      T     #OutTotalWeight;
      L     #Set001.RecipeNr;
      T     #OutRecipeNr;
      L     #Set001.Step;
      T     #OutLCStep;
//Reset old alarm flags with CmdFaultReset
      A     #Par.HelpFlags.OutFlagFaultResetDone;
      A     "SYS_Pulse1000ms";
      R     #Par.HelpFlags.OutFlagFaultResetDone;
      R     #Par.HelpFlags.OutFaultResetDone;
      S     #Par.HelpFlags.OutTestNewAlarm;
      L     0;
      L     #Set001.AlarmNr;
      ==I;
      =     #Par.HelpFlags.OutNoAlarm;
//  keep old alalrm number
      A     #Par.HelpFlags.OutNoAlarm;
      A     #Par.HelpFlags.OutRelevantFault;
      AN    #Par.HelpFlags.OutTestNewAlarm;
      AN    #InLocal;
      AN    #InManual;
      JC    rA1;
      T     #OutAlarmNr;
//--------------------------------------
//Calculate job weight on WtNotErasable
rA1:  L     #Set001.WtNotErasable;
//---  Init first, if old value < 0  ---
      L     #Par.OutNotErasableWeight;
      L     0;
      <D;
      JC    PgZ2;
//---  Calculate Weight ---
      L     #Set001.WtNotErasable;
      L     #Par.OutNotErasableWeight;
      -D;
      JM    PgZ1;
      JU    PgPo;
PgZ1: L     L#1000000000;	//[7.5] Overflow is 999999999
      +D;
      JM    PgZ2;	//[7.5]
PgPo: L     10000;	// Maximum change by relaod software
      >D;
      JC    PgZ2;
      TAK;
      L     #OutJobWeight;
      +D;
      T     #OutJobWeight;	//--> Total weight
PgZ2: L     #Set001.WtNotErasable;
      T     #Par.OutNotErasableWeight;
      JU    R11;	//[7.0]   
//===============================
//[7.0]--> LC Parameter 
//Reading dataset 11
R11:  L     "SYS_DirectCtrlLCDB".PC.ObjectNo;
      L     #Par.ParObjectNo;
      <>I;
      JC    R127;
      AN    "SYS_DirectCtrlLCDB".PC.Hsk.FExamineFirst;
      AN    "SYS_DirectCtrlLCDB".PC.Hsk.FExamineNext;
      JC    R127;
// -- Start Reading with Dataset 11
      L     11;
      T     #DPData.NrRcvDataSet;
      L     253;	//First
      A     "SYS_DirectCtrlLCDB".PC.Hsk.FExamineFirst;
      JC    rLC9;
      L     254;	//Next
rLC9: T     #DPData.IdxRcvDataSet;
      JU    rcv0;
//---Answer  dataset 11 ---
//---Answer  dataset 12 ---
r11:  L     #DPData.NrRcvDataSet;
      L     11;
      <>I;
      JC    rLCB;
// Answer Dataset 11
      L     '  ';
      T     "SYS_DirectCtrlLCDB".PC.Value[1];
      L     #DPData.Data[1];
      T     DB10.DBD 60;
      L     #DPData.Data[2];
      T     DB10.DBD 64;
      L     #DPData.Data[3];
      T     DB10.DBD 68;
      L     #DPData.Data[4];
      T     DB10.DBD 72;
      L     #DPData.IdxRcvDataSet;
      L     255;
      ==I;
      JC    rLCE;
      S     "SYS_DirectCtrlLCDB".GC.Set11Done;
      L     12;
      T     #DPData.NrRcvDataSet;
      L     0;
      T     #DPData.IdxRcvDataSet;
      JU    rcv0;	//--> Read dataset 12
// Answer Dataset 12
rLCB: L     #DPData.NrRcvDataSet;
      L     12;
      <>I;
      JC    r127;
      L     #DPData.Data[1];
      T     DB10.DBD 76;
      L     #DPData.Data[2];
      T     DB10.DBD 80;
      L     #DPData.Data[3];
      T     DB10.DBD 84;
      L     #DPData.Data[4];
      T     DB10.DBD 88;
      AN    "SYS_DirectCtrlLCDB".GC.Set11Done;
      JC    R127;
rLCE: L     12;
      CALL  "SYS_DirectCtrl";
      JU    R127;
//<--[7.0]
//===============================
//Answer  dataset 127
r127: L     #DPData.NrRcvDataSet;
      L     127;
      <>I;
      JC    r128;
      L     #DPData.Data[2];	//WtActual
      SRD   24;
      T     #tmpDecPoint;
      L     0;	//0 Decimal points == 1000gr
      ==I;
      L     1000;
      JC    rmul;
      L     #tmpDecPoint;
      L     1;	//1 Decimal points == 100gr
      ==I;
      L     100;
      JC    rmul;
      L     #tmpDecPoint;
      L     2;	//2 Decimal points == 10gr
      ==I;
      L     10;
      JC    rmul;
      L     1;	//3 Decimal points == 1gr
rmul: L     #DPData.Data[1];	//WtActual
      *D;
      T     #OutScaleWeight;
      JU    R128;
//===============================
//Answer  dataset 128
r128: L     #DPData.NrRcvDataSet;
      L     128;
      <>I;
      JC    r129;
      JU    R129;
//===============================
//Answer  dataset 129
r129: L     #DPData.NrRcvDataSet;
      L     129;
      <>I;
      JC    r136;
      S     #RecipeDiff.OutReadDone;
      R     #RecipeDiff.CmdRead;
      L     #DPData.Data[1];
      T     #DUMP.InDumpWeight;
      L     #DPData.Data[2];
      T     #DUMP.InFlowrateHighLimit;
      L     #DPData.Data[3];
      T     #DUMP.InFlowrateLowLimit;
      L     #DPData.Data[4];
      T     #DUMP.spare;
      JU    R001;
//===============================
//Answer  dataset 136
r136: L     #DPData.NrRcvDataSet;
      L     136;
      <>I;
      JC    R001;	// =no valide answer read dataset 001
      CALL  "SIEMENS_BLKMOV" (
           SRCBLK                   := #DPData.Data,
           RET_VAL                  := #tmpReturn,
           DSTBLK                   := #Set136);
      L     #RecipeDiff.InRecipeNr;
      L     #DPData.IdxRcvDataSet;
      ==I;
      JCN   R001;
      S     #RecipeDiff.OutReadDone;
      R     #RecipeDiff.CmdRead;
      L     #Set136.Density;
      T     #RecipeDiff.InOutDensity;
      L     #Set136.Factor;
      T     #RecipeDiff.InOutFactor;
      L     #Set136.AutoCorrFactor;
      T     #RecipeDiff.InOutAutoCorrFactor;
      L     #Set136.CutoffWt;
      T     #RecipeDiff.InOutCutoffWeight;
      JU    R001;
//===============================
//Read Dataset 001
R001: L     1;
      T     #DPData.NrRcvDataSet;
      L     0;
      T     #DPData.IdxRcvDataSet;
      A     #Par.HelpFlags.OutFaultResetDone;
      AN    "SYS_Pulse1000ms";
      S     #Par.HelpFlags.OutFlagFaultResetDone;
      JU    rcv0;
//===============================
//Read Dataset 127
R127: L     127;
      T     #DPData.NrRcvDataSet;
      L     0;
      T     #DPData.IdxRcvDataSet;
      JU    rcv0;
//===============================
//Read Dataset 128
R128: JU    R129;
      JU    rcv0;
//===============================
//Read Dataset 129
R129: AN    #RecipeDiff.CmdRead;
      ON    #Par.ParDUMP;
      JC    R136;
      L     129;
      T     #DPData.NrRcvDataSet;
      L     0;
      T     #DPData.IdxRcvDataSet;
      JU    rcv0;
//===============================
//Read Dataset 136
R136: AN    #RecipeDiff.CmdRead;
      O     #Par.ParDUMP;
      JC    R001;
      L     136;
      T     #DPData.NrRcvDataSet;
      L     #RecipeDiff.InRecipeNr;
      T     #DPData.IdxRcvDataSet;
rcv0: NOP   0;
      A     #Par.HelpFlags.OutComFaultRead;
      O     #Par.HelpFlags.OutComFaultSend;
      =     #OutComFault;
DP_A: NOP   0;
NETWORK
TITLE =  All State Init
      NOP   0;
//===Global Group Orders===
      A     "GCS7_Gr_OutManualOn";	//Gr.OutManualOn
      S     #InManual;
      A     "GCS7_Gr_OutManualOff";	//Gr.OutManualOff
      R     #InManual;
      A     #InManual;
      S     "GCS7_Gr_InManual";	//Gr.InManualMode
      A     "GCS7_Gr_OutFaultReset";	//Gr.OutOutFaultReset
      S     #CmdFaultReset;
//---Report is on---
      A     "GCS7_Gr_OutReportAll";	//Gr.OutReportAll
      O     #InReport;
      =     #tmpReport;
//---Local---
      A     #InLocal;
      AN    #InManual;
      =     #tmpLocalFault;
      A     #tmpLocalFault;
      O     #InHWStop;
      O     #InDPFault;
      =     #tmpLocal;
//---Enable---
// tmpOff
      AN    #InEnable;
      AN    #Par.ParManual;	// 2C: U -> UN
      A     #InManual;
      O;
      AN    #InEnable;
      AN    #InManual;
      O     #CmdOff;
      O     #tmpLocal;
      =     #tmpOff;
// Continue after Emptying
      A     #InOutRestdischargeScale;	//[4.2]
      O     #InOutRestdischargeBin;	//[4.2]
      AN    #InManual;	//[4.2]
      R     #CmdRefill;	//[4.2]
// Reset Restdischarge                  //[?.?]
      A     #CmdNewJob;
      O     #CmdOn;
      O     #tmpOff;
      O     #CmdRefill;
      R     #InOutRestdischargeBin;	//[4.0]
      A     #CmdNewJob;	//[5.0]
      O     #CmdOn;	//[5.0]
      O     #tmpOff;	//[PE]
      O     #CmdRefill;	//[5.0]
      R     #InOutRestdischargeScale;	//[4.0]//[5.0]
//---On---
      A     #CmdNext;
      AN    #InManual;
      O     #CmdOn;
      AN    #tmpOff;
      =     #tmpOn;
//---[4.0->] Sequence stop DUMP scale
      A     #InSeqStopDUMP;
      A     #Par.ParDUMP;
      AN    #Par.ParNoStep;
      =     #tmpSeqStopDUMP;	//[<-4.0]
//--- Init in local mode  
      AN    #tmpLocal;
      ON    #OutComFault;	//[7.2]
      JC    alJL;
//     R     #OutComFault   [6.2]
      L     0;
      T     #OutFlowrate;	//[4.0]
//--- recognice depot empty
alJL: NOP   0;
//---                                   /
      A     #Par.Status.EnableFeeding_Empty;
      O     #Par.Status.OutOfTolerance_LL;
      =     #OutDepotEmpty;
//[4.0->] event fully emptying DIFF scale after depot empty alarm     
      A     #InOutRestdischargeBin;
      AN    #Par.ParDUMP;
      A(;
      O     #Par.Status.EnableFeeding_Empty;
      O     #Par.Status.OutOfTolerance_LL;
      );
      S     #InOutRestdischargeScale;	//[<-4.0] Fully emptying DIFF scale
//--- Fault   
      LAR1  P##tmpFilter;
      L     #OutAlarmNr;
      +AR1;	//Pointer to #tmpFilter[OutAlarmNumber]
      L     #OutAlarmNr;
      L     0;
      <>I;
      AN    L [AR1,P#0.0];	//#tmpFilter[OutAlarmNumber]
      O;
      A     #Par.Status.SumFault;
      AN    #tmpFilter[0];
      =     #Par.HelpFlags.OutRelevantFault;
      A     #Par.HelpFlags.OutRelevantFault;
      O     #OutComFault;
      O     #OutWrongValue;
      O(;	//[6.2]
      AN    #Par.Status.RemoteControlDP;	//[6.2]
      AN    #Par.ParOPTO22;	//[6.2]
      );	//[6.2]
      AN    #tmpLocal;
      =     #tmpFault;
//---                                   //[?.?]
      SET;
      R     #tmpClearCmdFlag;
//--- New Job
      AN    #CmdNewJob;
      JC    alJ0;
      S     #tmpClearCmdFlag;
      R     #OutWeightCleared;
      S     #Par.HelpFlags.CmdNewValue;
      S     #Par.HelpFlags.CmdNewJob;
      S     #CmdNewValue;
      L     0;	//Clear
      T     #OutJobWeight;	//Total weight
alJ0: NOP   0;
//---New Value -----------
      L     #DUMP.InDumpWeight;
      L     0;
      <>I;
      A     #CmdNewValue;
      A     #Par.ParDUMP;
      S     #Par.HelpFlags.CmdSend129;
//--- Recipe
      A     #RecipeDiff.CmdRead;
      R     #RecipeDiff.OutReadDone;
      A     #RecipeDiff.CmdSend;
      R     #RecipeDiff.OutSendDone;
NETWORK
TITLE = Monitoring [6.0]
//Monitoring Time [6.0]
      A     #StStopped;
      O     #CmdFaultReset;
      R     #Par.HelpFlags.OutAlarmTimeOut;	//[6.0]
      AN    #StDosing;	//[6.0]
      AN    #StStarting;	//[6.0]
      O     #Par.ParDUMP;	//[6.0]
      JC    mtJ0;	//[6.0]
      L     #OutLCStep;	//[6.0]
      L     1;	//[6.0]
      >I;	//[6.0]
      O     #Par.ParNoStep;	//[6.0]
      O     #OutStopPoint;	//[6.0]
      JC    mtJ0;	//[6.0]
      ON    "GCS7_Gr_OutTick200ms";	//[6.0]
      JC    mtJ1;	//[6.0]
      L     #Par.OutMonTime;	//[6.0]
      +     -2;	//[6.0]
      T     #Par.OutMonTime;	//[6.0]
      L     0;	//[6.0]
      >=I;	//[6.0]
      JC    mtJ1;	//[6.0]
      S     #Par.HelpFlags.OutAlarmTimeOut;	//[6.0]
      JU    mtJ1;	//[6.0]
mtJ0: L     #Par.ParMonTime;	//[6.0]
      T     #Par.OutMonTime;	//[6.0]
mtJ1: NOP   0;
NETWORK
TITLE = States
//===State machine===
      A     #StStopped;
      JC    S0;
      A     #StStarting;
      JC    S1;
      A     #StDosing;
      JC    S2;
      A     #StEmptying;
      JC    S3;
      A     #StFault;
      JC    S4;
      A     #StEmptied;
      JC    S5;
      A     #StRefill;
      JC    S6;
      S     #StStopped;	//Init
NETWORK
TITLE = StStopped
//Transition to StStopped
//Transition
xxS0: S     #StStopped;
      JU    LOGX;
//----------------------------------------------
//Logic
//Condition for StFault
S0:   A     #tmpFault;
      R     #StStopped;
      JC    xxS4;
//StEmptying
      A     #InOutRestdischargeScale;
      O     #InOutRestdischargeBin;
      AN    #tmpSeqStopDUMP;	//[6.0]            
      A     #tmpOn;	//[6.0]
      R     #StStopped;
      JC    xxS3;
//StRefill
      A     #tmpOn;	//[7.4]
      AN    #Par.ParDUMP;
      A     #CmdRefill;
      R     #StStopped;
      JC    xxS6;
//Condition for StStarting
      A     #tmpOn;
      AN    #tmpSeqStopDUMP;	//[4.0]            
      R     #StStopped;
      JC    xxS1;
      JU    OUT;
NETWORK
TITLE =  STARTING
// Any Transition
//Transition
xxS1: S     #StStarting;
      S     #CmdNewValue;
      S     #tmpClearCmdFlag;
      JU    OUT;
//----------------------------------------------
//Logic
S1:   R     #OutEmptied;
      R     #OutRefillDone;
//Condition for StFault
      A     #tmpFault;
      O     #Par.HelpFlags.OutAlarmTimeOut;	//Monitoring Time [6.0]
      R     #StStarting;
      JC    xxS4;
//Condition for StStopped
      A     #tmpOff;
      O     #tmpSeqStopDUMP;	//[4.0]
      AN    #Par.ComFlags.S_Done;
      R     #StStarting;
      JC    xxS0;
//-- Transition to StDosing --         
      L     #OutLCStep;
      L     1;
      >I;
      O(;	//[6.4]
      A     #Par.Status.EnableFeeding_Empty;	//[6.4]
      A     #Par.ParDUMP;	//[6.4]
      );	//[6.4]    
      O     #Par.ParNoStep;
      A     #Par.Command.Start;
      O     #OutStopPoint;
      R     #StStarting;
      JC    xxS2;
      JU    OUT;
NETWORK
TITLE =  DOSING
//Transition
//----------------------------------------------
xxS2: SET;
      S     #StDosing;
      R     #Par.Status.Powerfailure;
      R     #OutWeightCleared;
      JU    LOGX;
//----------------------------------------------
//Condition for StEmptying
S2:   A     #InOutRestdischargeScale;
      O     #InOutRestdischargeBin;
      O;
      A     #InSeqStopDUMP;
      A     #Par.ParDUMP;
      R     #StDosing;
      JC    xxS3;
//Monitoring Time [6.0]
      A     #Par.HelpFlags.OutAlarmTimeOut;	//[6.0]
      R     #StStarting;	//[6.0]
      R     #StDosing;	//[6.0]
      JC    xxS4;	//[6.0]
//Condition for StStopped
//  Case 1 : DUMP , OPTO22
      A(;
      L     #OutLCStep;
      L     2;	//[6.5]
      <=I;
      O     #Par.ParNoStep;
      A     #Par.ParOPTO22;
      A     #Par.ParDUMP;	//[6.1]
//  Case 2 : DIFF , OPTO22
      O(;	//[6.1]
      L     #OutLCStep;	//[6.1]
      L     2;	//[6.1]
      <=I;	//[6.1]
      O     #Par.ParNoStep;
      A     #Par.ParOPTO22;
      AN    #Par.ParDUMP;	//[6.1]
      );	//[6.1]
//  Case 3 : Profibus
      O;
      AN    #Par.Status.Operation;	//[6.1]
      AN    #Par.ParOPTO22;	//[6.1]
//  All
      );	//[6.1]
      AN    #Par.Command.Start;
      A(;
      O     #tmpOff;
      ON    #OutStopPoint;
      );
      O;	//[6.2]
      A     #OutComFault;	//[6.2]
      AN    #tmpFault;	//[6.2]
      R     #StDosing;
      JC    xxS0;
//Condition for Fault
      A     #tmpFault;
      R     #StDosing;
      JC    xxS4;
      JU    OUT;
NETWORK
TITLE =  FAULT
//Condition for StStopped 
S4:   A     #Par.HelpFlags.OutTestNewAlarm;
      AN    #tmpFault;
      O     #tmpLocalFault;
      JC    S4S0;
      A     #Par.HelpFlags.OutTestNewAlarm;	//[2.3] Relog fault
      A     #tmpFault;	//[2.3]
      JC    xxS4;	//[2.3]
      JU    OUT;
//Transition to StStopped 
S4S0: S     #StStopped;
      R     #StFault;
      JU    LOG2;	//-->//Message ('fault cancelled')
NETWORK
TITLE =  StEmptying
//Transition
//----------------------------------------------
xxS3: S     #StEmptying;
      R     #OutEmptied;
      R     #OutRefillDone;
      R     #Par.HelpFlags.OutTargetSnd;	//[5.0]
      R     #Par.HelpFlags.OutStepRcv;	//[5.0]
      JU    OUT;
//----------------------------------------------
// Condition for fault
S3:   A     #tmpFault;
      R     #StEmptying;
      JC    xxS4;
//Condition for emptied
      L     #OutLCStep;	//Step 1 = Init
      L     1;
      ==I;
      A(;
      AN    #Par.ParDUMP;
      A(;
      A     #Par.Status.RestDischargeDone;
      A     #tmpMEAF;
      O;
      AN    #Par.Status.PreCutoffWt_ReadyDosing;
      AN    #tmpMEAF;
      A     #Par.HelpFlags.OutTargetSnd;
      A     #Par.HelpFlags.OutStepRcv;
      );
      O;
      A     #Par.ParDUMP;
      A     #Par.Status.RestDischargeDone;
      );
      A     #StEmptying;
      R     #StEmptying;
      JC    xxS5;	//-->StEmptied
//[4.0->] Back to Stopped if not empyting
      AN    #InSeqStopDUMP;
      ON    #Par.ParDUMP;
      AN    #InOutRestdischargeScale;
      AN    #InOutRestdischargeBin;
      R     #StEmptying;	//avoid setting of OutEmptied
      R     #InOutRestdischargeScale;
      JC    xxS1;	//[<-4.0]  [7.7] Change to StStarting
      JU    OUT;
NETWORK
TITLE =  StEmptied
//Condition for fault
//Transition
//----------------------------------------------
xxS5: S     #StEmptied;
      S     #OutEmptied;
      JU    LOGX;
//----------------------------------------------
S5:   A     #tmpFault;
      R     #StEmptied;
      JC    xxS4;
//Condition for Starting
      A     #InManual;
      A     #CmdOn;
      O;
      A     #Par.HelpFlags.CmdNewJob;
      AN    #InManual;
      R     #StEmptied;
      JC    xxS1;
//Condition for Stopped
      AN    #InOutRestdischargeScale;
      AN    #InOutRestdischargeBin;
      ON    #InEnable;
      R     #StEmptied;
      JC    xxS0;
      JU    OUT;
NETWORK
TITLE = StRefill
//Transition
xxS6: S     #StRefill;
      R     #OutEmptied;
      R     #OutRefillDone;
      JU    OUT;
//----------------------------------------------
//Condition for fault
S6:   A     #tmpFault;
      R     #StRefill;
      JC    xxS4;
//Condifition for StStopped
      A     #Par.Status.PreCutoffWt_ReadyDosing;
      ON    #CmdRefill;	//[5.0] PE
      R     #StRefill;
      R     #CmdRefill;
      S     #OutRefillDone;
      JC    xxS0;
      JU    OUT;
NETWORK
TITLE = LOG
////[5.0] Alarmnummer
xxS4: S     "GCS7_Gr_InFaultFlag";	//Gr.InFaultFlag
      S     #StFault;
//Horn On
      CALL  "SYS_Horn_Code" (
           FcCode                   := 1,
           ParObjectType            := 1040,
           ParObjectNo              := #Par.ParObjectNo,
           ParHornCode              := #Par.ParHornCode);
//Alarm Communication
      L     B#(1, 96);
      A     #OutComFault;
      JC    LOG;
//Tiemout
      A     #Par.HelpFlags.OutAlarmTimeOut;
      L     B#(1, 94);	// Message ('fault timeout')
      JC    LOG;
//Alarm-Nr 1..80
      L     0;
      L     #OutAlarmNr;
      ==I;
      JC    LOG1;
      L     B#(1, 0);
      OW;
      JU    LOG;	//Alarms 1..80
//Fault Remote Control
LOG1: L     B#(1, 90);	// Message ('fault DP Mode')   //[6.2]
      AN    #Par.Status.RemoteControlDP;	//[6.2]
      AN    #Par.ParOPTO22;	//[6.2]
      JC    LOG;	//[6.2]
//Wrong Value
      A     #OutWrongValue;
      L     B#(1, 95);	// Message ('fault wrong value')
      JC    LOG;
//Collected Alarm
      L     B#(1, 99);	// Message ('fault collected alarm')
      JU    LOG;
//Fault Canceled
LOG2: L     B#(4, 0);	// Message ('fault Fault Canceled')
      JU    LOG;
//===============================================
//State Transition
LOGX: AN    #tmpReport;
      JC    OUT;
      A     #StStopped;
      L     B#(4, 91);	//Message ('Stopped')
      JC    LOG;
      A     #StEmptied;
      L     B#(4, 92);	//Message ('Dosing')
      JC    LOG;
      A     #StEmptied;
      L     B#(4, 93);	//Message ('emptied')
      JC    LOG;
      JC    OUT;
LOG:  A     #Par.ParLogOff;	//---Set LOG Message
      JC    OUT;
      T     #tmpLOGvalue;
      L     W#16#FF;
      AW;
      T     #OutAlarmNrLog;
      CALL  "GCS7_LogConvert" (
           ObjectNo                 := #Par.ParObjectNo,
           MsgType                  := #Par.ParMsgType,
           ClassMsgTxt              := #tmpLOGvalue,
           OType                    := 1040);	//LOG Message Converter / Entry / Contains Class and TextNo
NETWORK
TITLE = Global End
OUT:  SET;	//---Clear commands
      R     #CmdNext;
      R     #CmdOn;
      R     #CmdNewJob;
      R     #Par.HelpFlags.OutTestNewAlarm;
      A     #StStopped;
      R     #CmdOff;
//=============================================
//OutStopPoint
//=============================================
//DIFF
      O     #Par.ParDUMP;
      O     #Par.HelpFlags.CmdNewValue;
      O     #CmdNewValue;
      JC    SAEE;
      A     #Par.Status.TotalReached;
      =     #OutStopPoint;
//DUMP
SAEE: ON    #Par.ParDUMP;
      O     #Par.HelpFlags.CmdNewValue;
      O     #CmdNewValue;
      JC    SAJ1;
      L     #InPreCutoffWeight;	//[4.0]
      L     #OutJobWeight;	//[4.0]
      +D;
      L     #InJobWeight;	//[4.0]
      >=D;
      O     #Par.Status.TotalReached;	//[7.8]
      =     #OutStopPoint;
SAJ1: NOP   0;
//--Output for group 
      A     #InDPFault;
      AN    #tmpLocalFault;
      S     "GCS7_Gr_InDPFault";
      A     #InHWStop;
      AN    #tmpLocalFault;
      S     "GCS7_Gr_InHWStop";
      A     #StFault;
      S     "GCS7_Gr_InFault";	// Gr.InFault
NETWORK
TITLE = Start / OutpEnable
      AN    #StEmptying;
      AN    #StStarting;
      AN    #StDosing;
      AN    #StRefill;
      O     #StStopped;
      O     #StFault;
      O     #tmpOff;
      O     #tmpSeqStopDUMP;
      O(;
      A     #StEmptying;
      O     #StRefill;
      AN    #Par.ParDUMP;
      A     #InOutRestdischargeScale;
      );
      O;
      A(;
      A     #Par.HelpFlags.CmdNewJob;
      AN    #tmpMEAF;
      );
      =     #tmpImmediateStop;
//  Set:
      AN    #tmpImmediateStop;
      AN    #Par.HelpFlags.CmdNewValue;
      AN    #CmdNewValue;
      AN    #Par.HelpFlags.CmdNewJob;
      S     #Par.Command.Start;
      S     #OutpEnable;
//  Reset:
      A     #InDisableDischargeDUMP;
      A     #Par.ParDUMP;
      O     #tmpImmediateStop;
      R     #OutpEnable;
      A     #StEmptying;
      A     #Par.ParDUMP;
      O     #tmpImmediateStop;
      R     #Par.Command.Start;
NETWORK
TITLE = Prepare Command for MEAF
      NOP   0;
//==============================
      A     #Par.Status.AcceptNewSendData;
      A     #Par.Command.ResetAlarm;
      AN    #Par.ParOPTO22;
      R     #Par.Command.ResetAlarm;
      S     #Par.HelpFlags.OutFaultResetDone;
      AN    #Par.Status.AcceptNewSendData;
      O     #Par.ParOPTO22;
      A     #CmdFaultReset;
      R     #CmdFaultReset;
      S     #Par.Command.ResetAlarm;
//==============================
      AN    #InDisableDischargeDUMP;
      A     #StEmptying;
      A     #Par.ParDUMP;
      O;
      A(;	//[6.6]
      L     #OutLCStep;	//[6.6]
      L     1;	//[6.6]
      ==I;	//[6.6]
      O     #Par.Command.RestDischarge;	//[6.6]
      );	//[6.6]
      A     #StEmptying;
      A     #InOutRestdischargeScale;
      AN    #Par.ParDUMP;
      =     #Par.Command.RestDischarge;
//================================
      A     #Par.Status.AcceptNewSendData;
      A     #Par.Command.ResetWtTotal;
      AN    #Par.ParOPTO22;
      S     #OutWeightCleared;
      R     #Par.Command.ResetWtTotal;
      R     #Par.HelpFlags.CmdNewJob;
      AN    #Par.Status.AcceptNewSendData;
      O     #Par.ParOPTO22;
      A     #Par.HelpFlags.CmdNewJob;
      S     #Par.Command.ResetWtTotal;
//==========================================================
//Restdosing/Refill
//===========================================================
//  --Restdosing 
      L     #OutLCStep;
      L     1;
      ==I;
      A     #Par.Status.PreCutoffWt_ReadyDosing;
      AN    #OutEmptied;
      A     #Par.Command.RestDischarge;
      O     #InRestDosing;
      A     #Par.ParDUMP;
      O;
//  --Refill 
      A     #StRefill;
      AN    #Par.ParDUMP;
      =     #Par.Command.RestDosing_Refill;
//==============================
      A     #InEnable;
      AN    #InDisableDischargeDUMP;
      AN    #InManual;	//[6.2]
      O;	//[6.2]
      A     #InManual;	//[6.2]
      AN    #StStopped;	//[6.2]
      AN    #StFault;	//[6.2]
      =     #Par.Command.EnableEmptying;
//==============================
      A     #InOutRestdischargeBin;
      AN    #Par.ParDUMP;
      =     #Par.Command.OverwriteLL;
//==============================
      A     #Par.Status.NewDataReady;
      =     #Par.Command.AcceptNewDataReady;
//==============================
      SET;
      =     #Par.Command.CommandReady;
//==============================
      A     #Par.Status.NewRcvData;
      =     #Par.Command.AcceptNewRcvData;
//==============================
      AN    #Par.Status.AcceptNewSendData;
      =     #Par.Command.NewSendData;
NETWORK
TITLE = (Profibus) Send Data
//**********************************
//(Profibus)
//**********************************
      A     #Par.ParOPTO22;
      JC    DP_C;
//======================================================
//Test Send Dataset 000 done
      L     #DPData.NrSndDataSet;
      L     0;
      <>I;
      JC    s128;
      JU    S128;	//-->send 128
//------------------------------------------------
//Test Send Dataset 128 done
s128: L     #DPData.NrSndDataSet;
      L     128;
      <>I;
      JC    s129;
      AN    #Par.Status.WrongValue;
      A     #Par.HelpFlags.CmdNewValue;
      A     #CmdNewValue;
      R     #Par.HelpFlags.CmdNewValue;
      R     #CmdNewValue;
      A     #Par.Status.WrongValue;
      =     #OutWrongValue;
      JU    S129;	//-->Send 129
//------------------------------------------------
//Test Send Dataset 129,136 done
s129: L     #DPData.NrSndDataSet;
      L     129;
      <>I;
      A(;
      L     #DPData.NrSndDataSet;
      L     136;
      <>I;
      );
      JC    S000;
      L     #DPData.IdxSndDataSet;
      L     #RecipeDiff.InRecipeNr;
      ==I;
      O     #Par.ParDUMP;
      JCN   S128;	//-->Send 128
      AN    #Par.Status.WrongValue;
      R     #RecipeDiff.CmdSend;
      =     #RecipeDiff.OutSendDone;
      R     #Par.HelpFlags.CmdSend129;
      A     #Par.Status.WrongValue;
      =     #RecipeDiff.OutWrongValue;
      JU    S128;	//-->Send 128
//==================================================
//Send Dataset 128
S128: A     #CmdNewValue;
      ON    #Par.Status.TotalReached;
      O;
      A     #InOutRestdischargeBin;
      AN    #Par.ParDUMP;
      JCN   S129;	//-->Send 129
      A     #CmdNewValue;
      =     #Par.HelpFlags.CmdNewValue;
      L     128;
      T     #DPData.NrSndDataSet;
      L     0;
      T     #DPData.IdxSndDataSet;
      L     #InFlowrate;
      T     #DPData.Data[1];
      A     #InOutRestdischargeBin;
      AN    #Par.ParDUMP;
      L     0;
      JC    S8g1;
      L     #InJobWeight;
S8g1: T     #DPData.Data[2];
      L     #InPreCutoffWeight;
      SLD   16;
      T     #DPData.Data[3];	//-->Byte 16/17
      L     #InRecipeNr;
      SLD   16;	//4.0
      T     #DPData.Data[4];	//-->Byte 21
      JU    Snd;
//======================================================
//Send Dataset 129
S129: A     #RecipeDiff.CmdSend;
      O     #Par.HelpFlags.CmdSend129;
      A     #Par.ParDUMP;
      JCN   S136;
      L     129;
      T     #DPData.NrSndDataSet;
      L     0;
      T     #DPData.IdxSndDataSet;
      L     #DUMP.InDumpWeight;
      T     #DPData.Data[1];
      L     #DUMP.InFlowrateHighLimit;
      T     #DPData.Data[2];
      L     #DUMP.InFlowrateLowLimit;
      T     #DPData.Data[3];
      L     #DUMP.spare;
      T     #DPData.Data[4];
      JU    Snd;
//======================================================
//Send Dataset 136
S136: AN    #Par.ParDUMP;
      A     #RecipeDiff.CmdSend;
      JCN   S000;
      L     136;
      T     #DPData.NrSndDataSet;
      L     #RecipeDiff.InRecipeNr;
      T     #DPData.IdxSndDataSet;
      L     #RecipeDiff.InOutDensity;
      T     #Set136.Density;
      L     #RecipeDiff.InOutFactor;
      T     #Set136.Factor;
      L     #RecipeDiff.InOutAutoCorrFactor;
      T     #Set136.AutoCorrFactor;
      L     #RecipeDiff.InOutCutoffWeight;
      T     #Set136.CutoffWt;
      CALL  "SIEMENS_BLKMOV" (
           SRCBLK                   := #Set136,
           RET_VAL                  := #tmpReturn,
           DSTBLK                   := #DPData.Data);
      JU    Snd;
//======================================================
//Send Dataset 0
S000: L     0;
      T     #DPData.NrSndDataSet;
      L     0;
      T     #DPData.IdxSndDataSet;
//======================================================
//Senden DP
Snd:  CALL  "SIEMENS_BLKMOV" (
           SRCBLK                   := #Par.Command,
           RET_VAL                  := #tmpReturn,
           DSTBLK                   := #DPData.StatusCommand);
      A     #InSimulation;
      JC    sSim;
      CALL  "SIEMENS_DPWR_DAT" (
           LADDR                    := #tmpAddr,
           RECORD                   := #DPData,
           RET_VAL                  := #tmpReturn);
      L     #tmpReturn;
      L     0;
      <>I;
      =     #Par.HelpFlags.OutComFaultSend;
      JU    sEnd;
//write to Simulation
sSim: R     #Par.HelpFlags.OutComFaultSend;
      A     "GCS7_Gr_SimDPtoImage";
      L     P#Q 0.0;
      JC    rDB2;
      OPN   "TEST_IOSimuliOutput";
      L     P#DBX 0.0;
rDB2: L     #Par.ParIOByteNr;
      SLD   3;
      +D;
      LAR1;
      L     #DPData.StatusCommand;
      T     D [AR1,P#0.0];
      L     #DPData.NrSndDataSet;
      T     B [AR1,P#4.0];
      L     #DPData.IdxSndDataSet;
      T     B [AR1,P#5.0];
      L     #DPData.NrRcvDataSet;
      T     B [AR1,P#6.0];
      L     #DPData.IdxRcvDataSet;
      T     B [AR1,P#7.0];
      L     #DPData.Data[1];
      T     D [AR1,P#8.0];
      L     #DPData.Data[2];
      T     D [AR1,P#12.0];
      L     #DPData.Data[3];
      T     D [AR1,P#16.0];
      L     #DPData.Data[4];
      T     D [AR1,P#20.0];
sEnd: NOP   0;
DP_C: NOP   0;
NETWORK
TITLE = (OPTO 22) Communication
//**********************************
//(OPTO22)
//**********************************
      AN    #Par.ParOPTO22;
      JC    O22X;
//============================================================
// Clear "OutComFlags
//============================================================
      LAR1  #tmpAddrOutComFlags;
      AN    #tmpClearCmdFlag;
      JC    COJ0;
      L     0;
      T     D [AR1,P#0.0];	//Clear flag of commands
COJ0: L     0;
      L     D [AR1,P#0.0];	//Clear flag of commands
      <>I;
      JC    COJ1;
//============================================================
// Start a new telegram cycle if OutComFlags=0
//============================================================
//-- Condition for new values 
      A     #CmdNewValue;
      AN    #Par.HelpFlags.CmdNewValue;
      R     #CmdNewValue;
      S     #Par.HelpFlags.CmdNewValue;
//************************************************************
//Cyclic functions
//================
//Send Next Telegram 
//===========================================================
//Test communication active
COJ1: A     DBX 50.0;	//COM.LC0.CmdPut ;
      O     DBX 50.1;	//COM.LC0.CmdGet ;
      JC    OUT0;
//Immediate stop              
      A     #Par.Command.Start;
      FN    #Par.HelpFlags.EnableDosing;
      JC    CmdA;	//--> Command 'S' or 'A'
//== Send New Values ========================================
//--
      AN    #Par.HelpFlags.CmdNewValue;
      AN    #Par.Status.Powerfailure;
      JC    CO_s;
//--COMMAND "M" : (only old)                                  
      AN    #Par.ComFlags.M_Done;
      AN    #Par.ParMEAF;
      JC    CmdM;
//-----------------------------------------------------
//--COMMAND "C"  : (only DUMP)                                  
      L     #DUMP.InDumpWeight;
      L     0;
      <>I;
      AN    #Par.ComFlags.CC_Done;
      A     #Par.ParDUMP;
      JC    CmdC;
//--
//Commands Only with flow control: DUMP same as MWEE
      L     #Par.OutScaleType;
      L     4;
      <>I;
      ON    #Par.ParDUMP;
      JC    CO_q;
//-----------------------------------------------------
//--COMMAND "U"  : (only DUMP)                                  
      AN    #Par.ComFlags.U_Done;
      JC    CmdU;
//-----------------------------------------------------
//--COMMAND "O" : (only DUMP)
      AN    #Par.ComFlags.O_Done;
      JC    CmdO;
//=====================================================
//--COMMAND "Q" : (only old)
CO_q: AN    #Par.ComFlags.Q_Done;
      AN    #Par.ParMEAF;
      JC    CmdQ;
//-----------------------------------------------------
//--COMMAND "S" : (only old)
CO_s: A     #Par.Status.Powerfailure;
      AN    #Par.ComFlags.S_Done;	//Reset power fault flag
      JC    CmdS;
//-----------------------------------------------------
//--Command "T" : (only old)
      A(;
      A     #StStopped;	//[4.0] send cleared emptying signal in state stopped
      AN    #OutEmptied;	//[4.0] 
      O     #StEmptying;
      O;
      A     #StRefill;
      );
      AN    #Par.ParDUMP;
      AN    #Par.ParMEAF;
      AN    #Par.ComFlags.TT_Done;
      JC    CmdT;	// only for DIFF Scale
//-----------------------------------------------------
//--Command "A" : MEAF
      AN    #Par.ComFlags.A_Done;	//Command "A" 
      A     #Par.ParMEAF;
      JC    CmdA;
//--Command "S" : not MEAF
      AN    #Par.ComFlags.S_Done;	//Command 'S'
      AN    #Par.ParMEAF;
      JC    CmdS;
//-----------------------------------------------------
//Command "h" : (MEAF)
      A     #Par.ParMEAF;
      AN    #Par.ComFlags.h_Done;
      JC    Cmdh;
//-----------------------------------------------------
//Command "t" : (all)
      L     #Par.OutScaleType;	// [5.0]
      L     0;	// [5.0]
      ==I;	// [5.0]
      A     #StStopped;
      AN    #Par.ComFlags.t_Done;
      JC    Cmdt;
//-----------------------------------------------------
//Command "r" : (only old)
      A     #Par.ParDUMP;
      AN    #Par.ParMEAF;
      AN    #Par.ComFlags.r_Done;
      JC    Cmdr;
//-----------------------------------------------------
//Command "c" : (only old)
      AN    #Par.ParMEAF;
      AN    #Par.ComFlags.c_Done;
      AN    #Par.ParNoStep;
      JC    Cmdc;
//-----------------------------------------------------
//Command "w" : (only old)
      AN    #Par.ParMEAF;
      AN    #Par.ComFlags.w_Done;	//Command "w"
      JC    Cmdw;
//-----------------------------------------------------
//Command "d" : (only old)
      AN    #Par.ParDUMP;
      AN    #Par.ParMEAF;	// [5.0]
      AN    #Par.ComFlags.d_Done;	//Command "d"
      JC    Cmdd;
//-----------------------------------------------------
//Command "f" : (only old)
      A     #Par.ParDUMP;
      AN    #Par.ParMEAF;	// [5.0]
      AN    #Par.ComFlags.f_Done;	//Command "f"
      JC    Cmdf;
//-----------------------------------------------------
//Command "g" : (only old)
      AN    #Par.ParMEAF;
      AN    #Par.ComFlags.g_Done;	//Command "g"
      JC    Cmdg;
//================================================  
//Init if all Telegrams are send
      R     #Par.HelpFlags.CmdNewValue;
      L     0;
      LAR1  #tmpAddrOutComFlags;
      T     D [AR1,P#0.0];	//Clear flag of commands
      JU    OUT0;
Cmdh: S     #Par.ComFlags.h_Done;
      L     'h';
      JU    GET;
Cmdc: S     #Par.ComFlags.c_Done;
      L     'c';
      JU    GET;
Cmdd: S     #Par.ComFlags.d_Done;
      L     'd';
      JU    GET;
Cmdf: S     #Par.ComFlags.f_Done;
      L     'f';
      JU    GET;
Cmdg: S     #Par.ComFlags.g_Done;
      L     'g';
      JU    GET;
Cmdt: S     #Par.ComFlags.t_Done;
      L     't';
      JU    GET;
Cmdr: S     #Par.ComFlags.r_Done;
      L     'r';
      JU    GET;
Cmdw: S     #Par.ComFlags.w_Done;
      L     'w';
      JU    GET;
CmdM: S     #Par.ComFlags.M_Done;
      L     'M';
      JU    PUT;
CmdO: S     #Par.ComFlags.O_Done;
      L     'O';
      JU    PUT;
CmdU: S     #Par.ComFlags.U_Done;
      L     'U';
      JU    PUT;
CmdQ: S     #Par.ComFlags.Q_Done;
      L     'Q';
      JU    PUT;
CmdS: S     #Par.ComFlags.S_Done;
      L     'S';
      JU    PUT;
CmdA: AN    #Par.ParMEAF;
      JC    CmdS;
      S     #Par.ComFlags.A_Done;
      L     'A';
      JU    PUT;
CmdT: S     #Par.ComFlags.TT_Done;
      L     'T';
      JU    PUT;
CmdC: S     #Par.ComFlags.CC_Done;
      L     'C';
      JU    PUT;
PUT:  S     DBX 50.0;	//COM.LC0.CmdPut ;
      JU    ALL1;
GET:  S     DBX 50.1;	//COM.LC0.CmdGet ;
ALL1: T     DBB 51;	//COM.LC0.Command;
OUT0: NOP   0;
O22X: NOP   0;
NETWORK
TITLE = State Code
//--Stopped, Substate ---
      AN    #StStopped;
      JC    STC2;
      L     41;	//Code: StStopped.HWStop
      A     #InHWStop;
      JC    STC;
      L     51;	//Code: StStopped.DPFault
      A     #InDPFault;
      JC    STC;
      L     1;	//Code: stopped
      A     #StStopped;
      JC    STC;
//===============
STC2: L     2;	//Code: starting
      A     #StStarting;
      JC    STC;
      L     3;	//Code: dosing
      A     #StDosing;
      JC    STC;
      L     9;	//Code: emptying
      A     #StEmptying;
      JC    STC;
      L     10;	//Code: emptied
      A     #StEmptied;
      JC    STC;
      L     11;	//Code: refill
      A     #StRefill;
      JC    STC;
      L     32;	//Code: fault
STC:  L     #StCode;	//Old state code
      TAK;
      T     #StCode;	//Save state code
      <>I;
      L     3;	//Load code for CBit methode
      CC    "SYS_CBitCtrl";
NETWORK
TITLE =  Store LC data
//**********************************
//(OPTO22)
//**********************************
      AN    #Par.ParOPTO22;
      BEC;
      L     #Par.ParLCIdx;
      T     DBW 34;	//COM.Element.Index; 
      L     2;	//Store LC data
      T     DBW 0;	//COM.CODE;
      CDB;
      UC    "GCS7_RS485Ctrl";
      CDB;
END_FUNCTION_BLOCK

FUNCTION_BLOCK "GCS7_M_MYFA"	// FB 41
TITLE = Machine MYFA
//  
//COPYRIGHT:    (C) 1997  BUHLER AG, CH-9240 UZWIL, SWITZERLAND
//
//PRODUCT:      GCS7
//
//TITLE:        FB 41 Machine  Control:Dampening with  MYFA/MOZD 
//                                     Produktbenetzung mit MYFA/MOZD
//
//-------------------------------------------------------------------------
//
//IDENT:        AUTHOR:             DEPT:                       DATE:
//
//FB41.5.2      A. Egli             CT3                         25-Jul-2007
//              Condition ParWithAirValue 
//FB41.5.1      A. Egli             CT3                         20-Feb-2006
//              For delay timer check ParWithAirValue
//FB41.5.0      A. Egli             CT3                         17-Jun-2002
//              New Release with one block 
//FB41.4.0      A.Egli              CT3                         06-Nov-2001
//              - ParOffDelayFeed ; -ParOnDelayWater             
//              !!! GCPROVB: Revision 40
//FB41.3.4      A.Egli              CT3                         05-Nov-2001
//              FlowWaterMin.InLocal
//              The ASW can program FlowWaterMin.InMonTrue if necessary.
//FB41.3.3      E.Hanselmann/A.Egli MU664/CT3                   25-Jan-2001
//              AirValve.InSeqStop correction
//              Transition StStarting-->StWait
//              Condition FlowProd.CmdRunTimeoutTime
//FB41.3.2      A.Egli              CT3                         09-Oct-2000
//              FlowProd.CmdRunTimeoutTime, 1 working condition for FlowProd
//FB41.3.1      S. Kalberer         CT3                         02-Oct-2000
//              ParFlowProdLocal added
//FB41.3.0      A. Egli             CT3                         11-Oct-1999
//              Local data reduced 
//FB41.2D       A. Egli             CT3                         13-Sep-1999
//              Possibility to monitor FlowProd
//FB41.2C       A. Egli             CT3                         27-Aug-1999
//              tmpStarted: Check if AirValve is used,tmpStopWater
//FB41.2B       K. Tischer          MU664                       06-Mrz-1999
//              CC FC2 not UC FC2
//FB41.2A       A. Egli             CT3                         04-Mai-1998
//              StFault = StCode 32
//FB41.1A       A.Egli              AEE61                       15-Oct-1997
//              1st Release in S7
//
//-------------------------------------------------------------------------
//
//PURPOSE:      MANUAL : see [LL.MZDxxMAN]
//
//RESTRICTIONS: S7
//              ACCU2: Pointer to dynamic datas of the machine
//              ACCU1: Pointer to parameter datas of the machine
//
//-------------------------------------------------------------------------
//
AUTHOR : EA
FAMILY : GCS7LL
NAME : MOZDMYFA
VERSION : 5.2
VAR
  Ma : UDT 20410;
  MYFAMOZD : FB 39;	//Element
  FlowWaterMin : FB 14;	//Element
  FlowWaterMax : FB 14;	//Element
  FlowProd : FB 14;	//Element
  HLInlet : FB 14;	//Element
  AirValve : FB 13;	//Element
  WaterValve : FB 13;	//Element
  BypassFlap : FB 13;	//Element
END_VAR
VAR_TEMP
  tmpEnable : BOOL ;
  tmpFault : BOOL ;
  tmpRemoteWaterControl : BOOL ;
  tmpManualWaterControl : BOOL ;
  tmpLocalWaterControl : BOOL ;
  tmpLocal : BOOL ;
  tmpStarted : BOOL ;
  tmpStopWater : BOOL ;
  tmpLenDyn : INT ;
  tmpStoreAR2 : DINT ;
END_VAR
BEGIN
NETWORK
TITLE =
      L     24;
      T     #tmpLenDyn;
NETWORK
TITLE = PC Control
//=== Test Object number =====================
      L     "SYS_DirectCtrlDB".PC.ObjectNo;	//PCControl.ObjectNo
      L     #Ma.Par.ParObjectNo;	//Input ObjectNo
      <>I;
      JC    aEnd;
//=== Test OType      ========================
      L     2041;	//Input object type
      L     "SYS_DirectCtrlDB".PC.ObjectType;	//PCControl.ObjectType
      <>I;
      JC    aEnd;
//=== Test Handshake =========================
      A     "SYS_DirectCtrlDB".PC.Hsk.FExamine;	// Handshake.FExamine
      JC    aExa;
      A     "SYS_DirectCtrlDB".PC.Hsk.FDefineCmd;	// Handshake.FDefineCmd
      JC    aCmd;
      A     "SYS_DirectCtrlDB".PC.Hsk.FDefinePara;	// Handshake.FDefinePara
      JC    pPar;
aIni: L     2;	// FcInit
      UC    "SYS_DirectCtrl";
      JU    aEnd;
// Write parameter 
pPar: LAR1  P#DBX 58.0;
      L     P#6.0;
      +AR1;
      L     DBW [AR1,P#4.0];
      T     #Ma.Par.ParOffDelayFeed;
      L     DBW [AR1,P#6.0];
      T     #Ma.Par.ParOnDelayWater;
// Write new commands from PC to Interface of group 
aCmd: A     "SYS_DirectCtrlDB".PC.Cmd1[8];	//Cmd1[8]=CmdOff
      S     #Ma.CmdOff;
      A     "SYS_DirectCtrlDB".PC.Cmd1[9];	//Cmd1[9]=CmdOn
      S     #Ma.CmdOn;
      A     "SYS_DirectCtrlDB".PC.Cmd1[2];	//Cmd1[2]=CmdLocalWaterControl
      S     #Ma.InLocalWaterControl;
      R     #Ma.InRemoteWaterControl;
      R     #Ma.InManualWaterControl;
      A     "SYS_DirectCtrlDB".PC.Cmd1[3];	//Cmd1[3]=CmdRemoteWaterControl
      R     #Ma.InLocalWaterControl;
      S     #Ma.InRemoteWaterControl;
      R     #Ma.InManualWaterControl;
      A     "SYS_DirectCtrlDB".PC.Cmd1[4];	//Cmd1[4]=CmdManualWaterControl
      R     #Ma.InLocalWaterControl;
      R     #Ma.InRemoteWaterControl;
      S     #Ma.InManualWaterControl;
      A     "SYS_DirectCtrlDB".PC.Cmd1[10];	//Cmd1[10]=CmdNext
      S     #Ma.CmdNext;
      A     "SYS_DirectCtrlDB".PC.Cmd1[11];	//Cmd1[11]=CmdFaultReset
      S     #Ma.CmdFaultReset;
      A     "SYS_DirectCtrlDB".PC.Cmd1[13];	//Cmd1[13]=CmdManualOn
      S     #Ma.InManual;
      A     "SYS_DirectCtrlDB".PC.Cmd2[13];	//Cmd2[13]=CmdManualOff
      R     #Ma.InManual;
      JU    aIni;
aExa: TAR2;	// Address Dynamic datas
      T     "SYS_DirectCtrlDB".GC.InDynAddr;	// -->PCControl.GC.InDynAddr
      L     #tmpLenDyn;	// Length Dynamic datas
      T     "SYS_DirectCtrlDB".GC.InDynLen;	// -->PCControl.GC.InDynLen
      L     0;
      T     "SYS_DirectCtrlDB".GC.InParaAddr;	// -->PCControl.GC.InParaAddr
      T     "SYS_DirectCtrlDB".GC.InParaLen;	// -->PCControl.GC.InParaLen
      L     1;	// Code FcExamine
      UC    "SYS_DirectCtrl";
      L     10;	//Revision
      T     "SYS_DirectCtrlDB".GC.Revision;
aEnd: NOP   0;
NETWORK
TITLE =  Timer switch off feed and switch on water  
//Timer switch off delay feed
//[4.0 --->
      A     #WaterValve.StHN;
      O     #AirValve.StHN;
      A     #Ma.OutReadyFeeding;
      AN    #Ma.InFeeding;
      JC    TiF0;
      R     #Ma.OutOffDelayFeedRun;
      L     0;	//Reset timervalue to zero
      T     #Ma.Par.OutOffDelayFeed;
      JU    TiW;
TiF0: A     #Ma.OutOffDelayFeedDone;
      JC    TiW;
      A     #Ma.OutOffDelayFeedRun;
      JC    TiF1;
      S     #Ma.OutOffDelayFeedRun;
      L     #Ma.Par.ParOffDelayFeed;
      T     #Ma.Par.OutOffDelayFeed;
TiF1: AN    "GCS7_Gr_OutTick1s";	//Gr.OutTick1S
      L     #Ma.Par.OutOffDelayFeed;
      JC    TiF2;
      +     -10;
      T     #Ma.Par.OutOffDelayFeed;
TiF2: L     0;
      <=I;
      R     #Ma.OutOffDelayFeedRun;
      S     #Ma.OutOffDelayFeedDone;
TiW:  A     #FlowProd.StTrue;
      O     #FlowProd.StCtoTrue;
      O     #FlowProd.InLocal;
      A(;
      A     #AirValve.StLN;	//[5.2]
      ON    #Ma.Par.ParWithAirValve;	//[5.2][5.1]
      A     #WaterValve.StLN;	//[5.2]
      );
      A     #Ma.OutReadyFeeding;
      A     #Ma.InFeeding;
      JC    TiW0;
      R     #Ma.OutOnDelayWaterRun;
      L     0;	//Reset timervalue to zero
      T     #Ma.Par.OutOnDelayWater;
      JU    TiE;
//Timer swtich on delay water
TiW0: A     #Ma.OutOnDelayWaterDone;
      JC    TiE;
      A     #Ma.OutOnDelayWaterRun;
      JC    TiW1;
      S     #Ma.OutOnDelayWaterRun;
      L     #Ma.Par.ParOnDelayWater;
      T     #Ma.Par.OutOnDelayWater;
TiW1: AN    "GCS7_Gr_OutTick1s";	//Gr.OutTick1S
      L     #Ma.Par.OutOnDelayWater;
      JC    TiW2;
      +     -10;
      T     #Ma.Par.OutOnDelayWater;
TiW2: L     0;
      <=I;
      R     #Ma.OutOnDelayWaterRun;
      S     #Ma.OutOnDelayWaterDone;
//---Reset timer Done bit
TiE:  A     #FlowProd.StFalse;
      AN    #FlowProd.InLocal;
      ON    #Ma.InFeeding;
      R     #Ma.OutOnDelayWaterDone;
      A     #Ma.InFeeding;
      R     #Ma.OutOffDelayFeedDone;
// <-- 4.0]
NETWORK
TITLE = Interlocking
//===Global Group Orders===
      A     "GCS7_Gr_OutManualOn";	///Gr.OutManualOn
      S     #Ma.InManual;
      A     "GCS7_Gr_OutManualOff";	//Gr.OutManualOff
      R     #Ma.InManual;
      A     #Ma.InManual;
      S     "GCS7_Gr_InManual";	//Gr.InManual
      AN    #Ma.InLocalWaterControl;
      A     #Ma.InRemoteWaterControl;
      AN    #Ma.InManualWaterControl;
      AN    #Ma.InLocalWaterControl;
      =     #tmpRemoteWaterControl;
      A     #Ma.InLocalWaterControl;
      AN    #Ma.InRemoteWaterControl;
      AN    #Ma.InManualWaterControl;
      =     #tmpLocalWaterControl;
      AN    #Ma.InLocalWaterControl;
      AN    #Ma.InRemoteWaterControl;
      A     #Ma.InManualWaterControl;
      =     #tmpManualWaterControl;
//Local
      A     #Ma.InLocal;
      AN    #Ma.InManual;
      =     #tmpLocal;
      A     #tmpLocal;
      =     #MYFAMOZD.InLocal;
      =     #HLInlet.InLocal;
      =     #FlowWaterMax.InLocal;
      =     #WaterValve.InLocal;
      =     #AirValve.InLocal;
      =     #BypassFlap.InLocal;
      =     #FlowWaterMin.InLocal;	//[4.0]
      A     #Ma.Par.ParFlowProdLocal;	//[3.1]
      AN    #tmpManualWaterControl;	//[3.1]
      O     #tmpLocal;	//[3.1]
      =     #FlowProd.InLocal;	//[2D]
//Enable 
      AN    #Ma.InLocal;
      O     #Ma.InManual;
      A     #Ma.InEnable;
      AN    #Ma.CmdOff;
      =     #tmpEnable;
      A     #tmpRemoteWaterControl;
      =     #MYFAMOZD.InRemote;
//New Job 
      A     #Ma.CmdNewJob;
      S     #MYFAMOZD.CmdNewJob;
      A     #MYFAMOZD.StFault;
      O     #FlowWaterMax.StFault;
      O     #FlowWaterMin.StFault;
      O     #HLInlet.StFault;
      O     #AirValve.StFault;
      O     #BypassFlap.StFault;
      O     #WaterValve.StFault;
      O     #FlowProd.StFault;	//[2D]
      =     #tmpFault;
      A     #tmpRemoteWaterControl;
      A     #MYFAMOZD.StStarted;
      A     #WaterValve.StLN;
      A(;
      O     #AirValve.StHN;
      ON    #Ma.Par.ParWithAirValve;
      );
      O;
      A     #tmpLocalWaterControl;
      A     #MYFAMOZD.StStopped;
      A     #WaterValve.StLN;
      A(;	//[2C]
      A     #AirValve.StHN;	//[2C]
      ON    #Ma.Par.ParWithAirValve;	//[2C] 
      );	//[2C]
      O;
      A     #tmpManualWaterControl;
      A(;
      O     #MYFAMOZD.StStopped;
      ON    #MYFAMOZD.Par.ParMYFA;
      );
      A     #WaterValve.StHN;
      A(;
      O     #AirValve.StLN;
      ON    #Ma.Par.ParWithAirValve;
      );
      =     #tmpStarted;
//General stopping condition
      CLR;	//[4.0]
      =     #WaterValve.InSeqStop;
      CLR;	//[4.0]
      =     #AirValve.InSeqStop;
      A     #FlowProd.StFalse;
      O     #FlowProd.StCtoFalse;	//[2C]
      O     #FlowProd.StFault;	//[2D]
      A(;
      O     #tmpManualWaterControl;
      ON    #Ma.Par.ParFlowProdLocal;	//[4.0]
//[4.0]   ON    #Ma.Par.ParWithMYFA      
      );
      ON    #tmpEnable;
      O     #MYFAMOZD.StFault;
      O     #FlowWaterMax.StFault;
      O     #FlowWaterMin.StFault;	//[4.0]
      O     #WaterValve.StFault;
      O     #AirValve.StFault;
      O     #BypassFlap.StFault;
      O(;
      AN    #Ma.OutOnDelayWaterDone;	//[4.0]
      AN    #AirValve.StHN;	//[4.0]
      AN    #WaterValve.StHN;	//[4.0]
      );
      O     #Ma.OutOffDelayFeedDone;	//[4.0]
      =     #tmpStopWater;
// Enable MOZD
      A     #tmpRemoteWaterControl;
      AN    #tmpStopWater;
      =     #MYFAMOZD.InEnable;
// Enable Water
      A     #tmpManualWaterControl;
      AN    #tmpStopWater;
      =     #WaterValve.InEnableHN;
// Enable Air
      A     #tmpRemoteWaterControl;
      O     #tmpLocalWaterControl;
      AN    #tmpStopWater;
      =     #AirValve.InEnableHN;
// Set manual flap
      A     #tmpManualWaterControl;
      =     #BypassFlap.InEnableHN;
//Set low position
      AN    #AirValve.InEnableHN;
      =     #AirValve.InEnableLN;
      AN    #WaterValve.InEnableHN;
      =     #WaterValve.InEnableLN;
      AN    #BypassFlap.InEnableHN;
      =     #BypassFlap.InEnableLN;
//Next
//[4.0]      U     #Ma.InFeeding
//[4.0]      U     #FlowProd.StTrue
//[4.0]      O(    
//[4.0]      UN    #tmpManualWaterControl
//[4.0]      U     #Ma.Par.ParWithMYFA
//[4.0]      )     
      AN    #Ma.StStopped;
      AN    #Ma.StFault;
      S     #MYFAMOZD.CmdNext;
      S     #BypassFlap.CmdNext;
      S     #AirValve.CmdNext;
      S     #WaterValve.CmdNext;
//Monitoring
      SET;
      S     #HLInlet.InMonFalse;
      S     #FlowWaterMax.InMonTrue;
      AN    #FlowProd.InMonTrue;	//[3.3]
      A     #Ma.InFeeding;	//[3.2][3.3]
      S     #FlowProd.CmdRunTimeoutTime;	//[3.2]      
      A     #Ma.InFeeding;	//[2D]
      =     #FlowProd.InMonTrue;	//[2D]
NETWORK
TITLE = Call MOZD
      CALL  #MYFAMOZD;	//FB39
NETWORK
TITLE = Call FlowWaterMin
      CALL  #FlowWaterMin;
NETWORK
TITLE = Call FlowWaterMax
      CALL  #FlowWaterMax;
NETWORK
TITLE = Call FlowProd
      CALL  #FlowProd;
NETWORK
TITLE = Call HLInlet
      AN    #Ma.Par.ParWithHLInlet;
      JC    E6;
      CALL  #HLInlet;
NETWORK
TITLE = Call WaterValve
E6:   CALL  #WaterValve;
NETWORK
TITLE = Call AirValve
      AN    #Ma.Par.ParWithAirValve;
      JC    E8;
      CALL  #AirValve;
NETWORK
TITLE = Call BypassFlap (MYFA)
E8:   AN    #Ma.Par.ParWithBypassFlap;
      JC    StJ0;
      CALL  #BypassFlap;
NETWORK
TITLE = Jump to actual state
StJ0: A     #Ma.StStopped;
      JC    S0;
      A     #Ma.StStarting;
      JC    S1;
      A     #Ma.StStarted;
      JC    S2;
      A     #Ma.StWaiting;
      JC    S6;
      A     #Ma.StFault;
      JC    S4;
      A     #Ma.StStopping;
      JC    S3;
NETWORK
TITLE = Stopped
//any Transition 
xxS0: S     #Ma.StStopped;	// ===> Initialisation
      JU    OUT;
//=== Logic
//Condition to StFault
S0:   A     #tmpFault;
      R     #Ma.StStopped;
      JC    xxS4;	//--> StFault
//Condition to StStarting
      AN    #MYFAMOZD.StStopped;
      ON    #WaterValve.StLN;
      O(;	//[2C]
      AN    #AirValve.StLN;
      A     #Ma.Par.ParWithAirValve;	//[2C] 
      );	//[2C]
      A     #Ma.InFeeding;	//[3.3]
      R     #Ma.StStopped;
      JC    xxS1;	//-->StStarting
//Condition to StWaiting
      A     #Ma.CmdNext;
      AN    #Ma.InManual;
      O     #Ma.CmdOn;
      A     #tmpEnable;
      R     #Ma.StStopped;
      JC    xxS6;	//-->StWaiting
      JU    OUT;
NETWORK
TITLE = StStarting
//any Transition 
xxS1: S     #Ma.StStarting;
//=== Logic
//Condition to StFault
S1:   A     #tmpFault;
      R     #Ma.StStarting;
      JC    xxS4;	//--> StFault
//Condition to StStarted
      A     #tmpStarted;
      R     #Ma.StStarting;
      JC    xxS2;	//--> StStarted
//Condition to StStopping
      AN    #MYFAMOZD.StStarted;
      AN    #WaterValve.StHN;
      AN    #AirValve.StHN;
      ON    #tmpEnable;
      R     #Ma.StStarting;
      JC    xxS3;	//--> StStopping
      AN    #Ma.InFeeding;	//[3.3]
      R     #Ma.StStarting;	//[3.3]
      JC    xxS6;	//--> StWaiting [3.3]
      JU    OUT;
NETWORK
TITLE = StStarted
//any Transition 
xxS2: S     #Ma.StStarted;
//=== Logic
//Condition to StFault
S2:   A     #tmpFault;
      R     #Ma.StStarted;
      JC    xxS4;	//--> StFault
//Condition to StStopping
      AN    #tmpStarted;
      AN    #tmpEnable;
      R     #Ma.StStarted;
      JC    xxS3;	//--> StStopping
//Condition to StWaiting
      AN    #tmpStarted;
      R     #Ma.StStarted;
      JC    xxS6;	//--> StWaiting
      JU    OUT;
NETWORK
TITLE = StWaiting
//any Transition 
xxS6: S     #Ma.StWaiting;
//=== Logic
//Condition to StFault
S6:   A     #tmpFault;
      R     #Ma.StWaiting;
      JC    xxS4;	//--> StFault
//Condition to StStarted
      A     #tmpStarted;
      R     #Ma.StWaiting;
      JC    xxS2;	//--> StStarted
//Condition to StStopped
      AN    #tmpEnable;
      R     #Ma.StWaiting;
      JC    xxS3;	//--> StStopping
      JU    OUT;
NETWORK
TITLE = StStopping
//any Transition 
xxS3: S     #Ma.StStopping;
//=== Logic
//Condition to StFault
S3:   A     #tmpFault;
      R     #Ma.StStopping;
      JC    xxS4;	//--> StFault
//Condition to StStopped
      AN    #MYFAMOZD.StStarted;
      AN    #WaterValve.StHN;
      AN    #AirValve.StHN;
      O(;
      A     #Ma.CmdNext;
      AN    #Ma.InManual;
      O     #Ma.CmdOn;
      A     #tmpEnable;
      );
      R     #Ma.StStopping;
      JC    xxS0;	//--> StStopped
      JU    OUT;
NETWORK
TITLE = StFault
//any Transition 
xxS4: S     #Ma.StFault;
//=== Logic
//Condition to StStopping
S4:   AN    #tmpFault;
      R     #Ma.StFault;
      JC    xxS3;	//--> StStopping
      JU    OUT;
NETWORK
TITLE = State Code
// State           StCode
// ----------------------
// StFault           32
// StStopped          1
// StStarting         2
// StStarted          3
// StWaiting          4
// StStopping         7
OUT:  A     #Ma.StFault;
      L     32;	//Code=Fault
      JC    Code;
      A     #Ma.StStopped;
      L     1;	//Code=Stopped
      JC    Code;
      L     2;	//Code=Starting
      A     #Ma.StStarting;
      JC    Code;
      L     3;	//Code=Started
      A     #Ma.StStarted;
      JC    Code;
      L     4;	//Code=Feeding
      A     #Ma.StWaiting;
      JC    Code;
      L     7;	//Code=Stopping
Code: L     #Ma.StCode;	// Old state code
      TAK;
      T     #Ma.StCode;	// Save state code
      <>I;
      L     3;
      CC    "SYS_CBitCtrl";	//Set change bit
// 
NETWORK
TITLE = Global End
      A     #Ma.CmdFaultReset;
      S     #MYFAMOZD.CmdFaultReset;
      S     #FlowWaterMin.CmdFaultReset;
      S     #FlowWaterMax.CmdFaultReset;
      S     #AirValve.CmdFaultReset;
      S     #BypassFlap.CmdFaultReset;
      S     #HLInlet.CmdFaultReset;
      S     #FlowProd.CmdFaultReset;
//---Output commands
      AN    #HLInlet.StFault;
      AN    #BypassFlap.StFault;
      =     #Ma.OutReadyFeeding;
//---Clear all commands
      CLR;
      =     #Ma.CmdOn;
      =     #Ma.CmdOff;
      =     #Ma.CmdNext;
      =     #Ma.CmdFaultReset;
      =     #Ma.CmdNewJob;
END_FUNCTION_BLOCK

FUNCTION_BLOCK "GCS7_E_BSPB"	// FB 42
TITLE = BSPB Topwhite Vertical Whitener
//  
//COPYRIGHT:    (C) 1997 BY  BUHLER AG, CH-9240 UZWIL  SWITZERLAND
//
//PRODUCT:      GCS7
//
//TITLE:        Element BSPB Topwhite Vertical Whitener (Profibus and Opto22)
//
//-------------------------------------------------------------------------
//
//IDENT:        AUTHOR:             DEPT:                      DATE:
//
//FB42.4.2      A. Egli             BASE                       09-Apr-2008
//              Disable Alarm 18 Battery Low
//FB42.4.1      A.Egli              CT3                        01-Dec-2005
//              Parameter Upload Change DBD86-->DBD88
//FB42.4.0      A.Egli              CT3                        05-Jan-2005
//              Parameter Upload (uses DB10)
//FB42.3.3      A. Egli             CT3                        13-Oct-2004
//              Profibus Interface
//FB42.3.2      G. Shingler         CDDP                       18-Dec-2003
//              Target value is now motor current, not Press%
//              Current and Press% swapped over in reply telegrams
//              Status reply bits corrected
//FB42.3.1      G. Shingler         CDDP                       26-Nov-2003
//              Correction to read values
//FB42.3.0      A. Egli             CT3                        07-Nov-2003
//              Recipe Number sent to BSPB
//FB42.2.0      A. Egli             CT3                        09-Okt-2003
//              Recipe Parameter sent to BSPB
//FB42.1.0      A. Egli             CT3                        08-Sep-2003
//              1st Release in S7
//
//-------------------------------------------------------------------------
//
//PURPOSE:      MANUAL : see [BSPBxxMAN]
//
//RESTRICTIONS: S7
//              ACCU2: Pointer to dynamic datas of the element
//              ACCU1: Pointer to parameter datas of the element
//
//=======================================================
//Log Message: 
//------------------------------------------------------
//0     = Fault Cannceled
//1..79 = AlarmLC : Alarmnumber see manual of MEAF
//91    = StStopped
//92    = StDosing
//93    = StEmptied
//94    = Timeout starting
//95    = Wrong value
//96    = Communication fault
//97    = 
//98    = 
//99    = Collected alarm
//
//=======================================================
//StCode:  State               
//------------------------------------------------------
//32    StFault                 
// 1    StStopped                   Stopped
//41    Stopped.HWStop              StStopped + InHWStop 
//51    Stopped.DPFault             StStopped + DPFault
// 2    StStarting              
// 3    StStarted               
// 7    StStopping              
//
//
AUTHOR : EA
FAMILY : GCS7LL
NAME : BSPB
VERSION : 4.2
VAR
  StCode : INT ;	//Element state code
  InEnable : BOOL ;	//Enable to run the element (manual and automatic mode)
  spare21 : BOOL ;
  spare22 : BOOL ;
  CmdNewValue : BOOL ;	//Send new target values
  spare0204 : BOOL ;
  spare0205 : BOOL ;
  spare0206 : BOOL ;
  spare0207 : BOOL ;
  CmdOff : BOOL ;	//Pulse to stop the element (manual mode)
  CmdOn : BOOL ;	//Pulse to start the element (manual mode)
  CmdNext : BOOL ;	//Pulse to start the element in automatic mode
  CmdFaultReset : BOOL ;	//Command to reset fault
  InLocal : BOOL ;	//1= Local mode (no fault by start with service switch)
  InManual : BOOL ;	//1= Manual / 0= Automatic
  InReport : BOOL ;	//Report of all state transitions
  spare0307 : BOOL ;
  InHWStop : BOOL ;	//HW stop is detected, no fault
  InDPFault : BOOL ;	//DP-Fault is detected, no fault
  InSimulation : BOOL ;	//BSPB: Simulation with DPSim
  OutComFault : BOOL ;	//Communication fault
  spare0404 : BOOL ;
  spare0405 : BOOL ;
  spare0406 : BOOL ;
  OutpEnable : BOOL ;	//Digital output dosing enable (only Opto22)
  StStopped : BOOL ;	//Element is stopped
  StStarting : BOOL ;	//Element is starting
  StStarted : BOOL ;	//Element is dosing
  StStopping : BOOL ;	//Element is stopping
  StFault : BOOL ;	//Element has a communication or device fault
  spare55 : BOOL ;
  spare56 : BOOL ;
  spare57 : BOOL ;
  OutWrongValue : BOOL ;	//Wrong nominal values, rejected by MEAF
  InMotorCurrent : DINT ;	//Nominal Motor Current [A]
  InRecipeNr : INT ;	//BSPB: Is send to LC
  spare14 : INT ;	//
  OutCurrentMotorNom : INT ;	//Is read from MEAF: Motor current [A]
  OutPressure : DINT ;	//Is read from MEAF: actual Pressuret [0.1%]
  OutScaleWeight : DINT ;	//Is read from MEAF: Scale weight [g]
  OutCurrentMotorAc : INT ;	//Is read from MEAF: Motor current [A]
  OutPMin : INT ;	//Is read from MEAF: min. Pressure [0.1%]
  OutPMax : INT ;	//Is read from MEAF: max. Pressure [0.1%]
  OutRecipeNr : INT ;	//Is read from MEAF: Recipe number
  OutLCStep : INT ;	//Is read from MEAF: Step number
  spare36 : INT ;	//
  spare38 : INT ;	//
  spare40 : INT ;	//
  spare42 : INT ;	//
  spare44 : INT ;	//
  spare46 : INT ;	//
  spare48 : INT ;	//
  spare50 : INT ;
  OutAlarmNr : INT ;	//Is read from MEAF
  OutAlarmNrLog : INT ;	//Last textnumber send to log
  Par : STRUCT
   ParObjectNo : INT ;	//Is used for communication with PC, e.g. for message
   ParMsgType : INT ;	//Is used for message (translation of state)
   ParHornCode : INT ;	//Is used by horn module
   ParLogOff : BOOL ;	//Report is off
   ParManual : BOOL ;	//Manual mode wihout interlocking
   ParOpto22 : BOOL ;	//1=OPTO22 communication, 0=DP
   ParFilter : STRUCT 	//Filter to alarm 1=Ignore alarm
    SumFault : BOOL ;	//All: de: Sammelalarm
    A05_24VToLow : BOOL ;	//All:
    A07ADRange : BOOL ;
    A08ADCalibration : BOOL ;
    A09ADFunction : BOOL ;
    A10ADSupply : BOOL ;
    A11AnalogInput : BOOL ;
    AxxCommunication : BOOL ;	//A12: Serial Interface ; A14=DPFault
    A13RemoteControl : BOOL ;
    A16Printer : BOOL ;
    A26Tolerance : BOOL ;
    A30ZeroTara : BOOL ;
    A38Slide : BOOL ;
    A39AirPressure : BOOL ;
    A46AutoRestart : BOOL ;
   END_STRUCT ;
   ParComDB : INT ;	//OPTO22  : Communication DB
   ParLCIdx : INT ;	//OPTO22  : Index of data record
   ParLCAddr : INT ;	//OPTO22  : Address of LC
   ParIOByteNr : INT ;	//PROFIBUS: Address of first input and output byte
   ParMonTime : INT ;	//Monitoring time starting and stopping
   OutMonTime : INT ;	//Monitoring time starting and stopping
   OutHelpFlags : STRUCT 	//Is sent to BSPB
    OutAlarmTimeOut : BOOL ;
    CmdNewValue : BOOL ;
    CmdFaultReset : BOOL ;
    OutFaultResetDone : BOOL ;
    OutTestNewAlarm : BOOL ;	//Aux. signal to retry fault message
    OutRelevantFault : BOOL ;
    OutNoAlarm : BOOL ;	//Alarmnumber 0 is read form LC
    OutFlagFaultResetDone : BOOL ;
    OutComFaultRead : BOOL ;
    OutComFaultSend : BOOL ;
   END_STRUCT ;
   Command : STRUCT
    Start : BOOL ;	//de: Start
    spare01 : BOOL ;
    spare02 : BOOL ;
    spare03 : BOOL ;
    spare04 : BOOL ;
    spare05 : BOOL ;
    spare06 : BOOL ;
    AcceptNewDataReady : BOOL ;	//BSPB: de: Quittierung neue Werte Bereit
    spare10 : BYTE ;
    spare20 : BYTE ;
    CommandReady : BOOL ;	//de: Steuersignale gültig
    spare31 : BOOL ;
    spare32 : BOOL ;
    spare33 : BOOL ;
    spare34 : BOOL ;
    ResetAlarm : BOOL ;	//de: Alarm löschen
    NewSendData : BOOL ;	//de: Aenderung Sendedaten
    AcceptNewRcvData : BOOL ;	//de: Quittierung Aenderung Empfangsdatensatz
   END_STRUCT ;
   Status : STRUCT
    Operation : BOOL ;	//de: Betrieb
    Startup : BOOL ;	//0=Startup done  , 1= Startup
    WarningHLC : BOOL ;	//1=Warning motor current > HLC
    InPosition : BOOL ;	//de: Stauteller in Position
    LevelProduct : BOOL ;	//Level product covered
    spare05 : BOOL ;
    spare06 : BOOL ;
    NewDataReady : BOOL ;	//de: Neue Werte Bereit
    spare10 : BOOL ;
    spare20 : BYTE ;
    spare30 : BOOL ;
    spare31 : BOOL ;
    spare32 : BOOL ;
    RemoteControl : BOOL ;	//de: Sollwertvorgabe Remote
    WrongValue : BOOL ;	//de: Falscher Sollwert
    SumFault : BOOL ;	//de: Sammelalarm
    AcceptNewSendData : BOOL ;	//de: Quittierung Aenderung Sendedaten
    NewRcvData : BOOL ;	//de: Aenderung Empfangsdaten
   END_STRUCT ;
  END_STRUCT ;
END_VAR
VAR_TEMP
  tmpLOGvalue : WORD ;	//LOG value
  tmpCommand : INT ;
  tmpFBNO : INT ;	//Number of the actual FB
  tmpFault : BOOL ;
  tmpOff : BOOL ;
  tmpOn : BOOL ;
  tmpLocal : BOOL ;
  tmpLocalFault : BOOL ;
  tmpReport : BOOL ;
  tmpFlag : BOOL ;
  tmpOutLCAlarmBinEmpty : BOOL ;
  tmpLenDyn : DINT ;
  tmpWt : DINT ;
  tmpFilter : ARRAY  [0 .. 100 ] OF BOOL ;
  tmpComDB : INT ;
  tmpStatus_h : STRUCT 	//Is read from BSPB
   Startupdone : BOOL ;
   Level : BOOL ;
   WarningHLC : BOOL ;
   SumFault : BOOL ;	//*3.2* Summary fault
   Remote : BOOL ;	//*3.2* BSPB is in remote
   NewValue : BOOL ;	//*3.2* BPSB received new data
   Operation : BOOL ;	//*3.2* BSPB in operation
   InPosition : BOOL ;	//*3.2* BSPB in target position
  END_STRUCT ;
  tmpCommand_A : STRUCT
   Start : BOOL ;
   Stop : BOOL ;
   Z0_1 : BOOL ;
   AlarmReset : BOOL ;
   Z1 : BYTE ;
   Z2 : BYTE ;
   Z3_0 : BOOL ;
   Z3_1 : BOOL ;
   Z3_2 : BOOL ;
   Modify : BOOL ;
  END_STRUCT ;
  tmpAddr : WORD ;
  tmpReturn : INT ;
  DPData : STRUCT
   StatusCommand : DWORD ;
   NrSndDataSet : BYTE ;	//de: Nummer Sendedatensatz
   IdxSndDataSet : BYTE ;	//de: Index Sendedatensatz
   NrRcvDataSet : BYTE ;	//de: Nummer Empfangsdatensatz
   IdxRcvDataSet : BYTE ;	//de: Index Empfangsdatensatz
   Data : ARRAY  [1 .. 4 ] OF DINT ;
  END_STRUCT ;
  Set001 : STRUCT
   CurrentMotorNom : INT ;	//Is read from MEAF: Motor current nominal [A]
   CurrentMotorAc : INT ;	//Is read from MEAF: Motor current actual [A]
   Pressure : INT ;	//Is read from MEAF: actual Pressuret [0.1%]
   PMin : INT ;	//Is read from MEAF: min. Pressure [0.1%]
   PMax : INT ;	//Is read from MEAF: max. Pressure [0.1%]
   spare18 : INT ;
   spare20 : BYTE ;
   RecipeNr : BYTE ;	//Is read from MEAF: Recipe number
   Step : BYTE ;
   AlarmNr : BYTE ;
  END_STRUCT ;
END_VAR
BEGIN
NETWORK
TITLE =  Start Global
      L     42;
      T     #tmpFBNO;
      L     88;
      T     #tmpLenDyn;	//--> Len dynamic data in byte
      L     #Par.ParComDB;
      T     #tmpComDB;
NETWORK
TITLE = Filter
      LAR1  P##tmpFilter;
      L     0;
      T     LD [AR1,P#0.0];	//tmpFilter[00..31]
      T     LD [AR1,P#4.0];	//tmpFilter[32..63]
      T     LD [AR1,P#8.0];	//tmpFilter[64..95]
      A     #Par.ParFilter.SumFault;
      =     #tmpFilter[0];
      A     #Par.ParFilter.A05_24VToLow;
      =     #tmpFilter[5];
      A     #Par.ParFilter.A07ADRange;
      =     #tmpFilter[7];
      A     #Par.ParFilter.A08ADCalibration;
      =     #tmpFilter[8];
      A     #Par.ParFilter.A09ADFunction;
      =     #tmpFilter[9];
      A     #Par.ParFilter.A10ADSupply;
      =     #tmpFilter[10];
      A     #Par.ParFilter.A11AnalogInput;
      =     #tmpFilter[11];
      A     #Par.ParFilter.AxxCommunication;
      =     #tmpFilter[12];
      =     #tmpFilter[14];	//[1.4]
      A     #Par.ParFilter.A13RemoteControl;
      =     #tmpFilter[13];
      A     #Par.ParFilter.A16Printer;
      =     #tmpFilter[16];
      SET;
      =     #tmpFilter[18];	//[4.2] Battery Low
      A     #Par.ParFilter.A26Tolerance;
      =     #tmpFilter[26];
      A     #Par.ParFilter.A30ZeroTara;
      =     #tmpFilter[30];
      A     #Par.ParFilter.A38Slide;
      =     #tmpFilter[38];
      A     #Par.ParFilter.A39AirPressure;
      =     #tmpFilter[39];
      A     #Par.ParFilter.A46AutoRestart;
      =     #tmpFilter[46];
NETWORK
TITLE = (Opto22) Call back function
//*****This functions are called by FBxxx (COM) ******
      AN    #Par.ParOpto22;
      JC    O22Z;
      OPN   DB [#tmpComDB];
      L     0;
      L     DBW 32;	//COM.Element.CODE;
      ==I;
      JC    PC;
      L     DBB 76;	//COM.Telegram.Command;
      T     #tmpCommand;
      L     1;
      L     DBW 32;	//COM.Element.CODE;
      ==I;
      JC    Send;
      L     2;
      ==I;
      JC    Rcv;
      L     4;	//NAK
      L     DBW 32;	//COM.Element.CODE;
      ==I;
      S     #OutComFault;	//fault communication
      JU    STOR;
//======================================================================
//Prepare Send Data 
//======================================================================
//--------------------
//Send A [3.1]
//--------------------
Send: L     #tmpCommand;
      L     'A';
      <>I;
      JC    SndZ;
      LAR1  P##tmpCommand_A;
      L     0;
      T     LD [AR1,P#0.0];	//-->Reset tmpStateTarget
//command 1
      A     #Par.Command.Start;
      =     #tmpCommand_A.Start;
      AN    #Par.Command.Start;
      =     #tmpCommand_A.Stop;
      A     #Par.Command.ResetAlarm;
      =     #tmpCommand_A.AlarmReset;
      SET;
      =     #tmpCommand_A.Modify;
      L     0;	//Character offset
      T     DBW 40;	//COM.Element.AddrOffset
      LAR1  P##tmpCommand_A;
      L     LB [AR1,P#0.0];
      T     DBD 36;	//COM.Element.InOutValue
      L     31;	//Convert Hex to 1-ASCII
      T     DBW 0;	//COM.CODE
      CDB;	//ComDB->Instanz-DB
      UC    "GCS7_RS485Ctrl";	//Convert (CODE=DBW0)
      CDB;	//ElementDB->Instanz-DB
// n.b    
      L     1;	//Character offset
      T     DBW 40;	//COM.Element.AddrOffset
      L     0;
      T     DBD 36;	//COM.Element.InOutValue
      L     32;	//Convert Hex to 1-ASCII
      T     DBW 0;	//COM.CODE
      CDB;	//ComDB->Instanz-DB
      UC    "GCS7_RS485Ctrl";	//Convert (CODE=DBW0)
      CDB;	//ElementDB->Instanz-DB
// Command 2    
      L     2;	//*3.2* Character offset
      T     DBW 40;	//COM.Element.AddrOffset
      LAR1  P##tmpCommand_A;
      L     LB [AR1,P#3.0];
      T     DBD 36;	//COM.Element.InOutValue
      L     31;	//Convert Hex to 1-ASCII
      T     DBW 0;	//COM.CODE
      CDB;	//ComDB->Instanz-DB
      UC    "GCS7_RS485Ctrl";	//Convert (CODE=DBW0)
      CDB;	//ElementDB->Instanz-DB
// Spare    
      L     3;	//*3.2* Character offset
      T     DBW 40;	//COM.Element.AddrOffset
      L     0;
      T     DBD 36;	//COM.Element.InOutValue
      L     31;	//Convert Hex to 1-ASCII
      T     DBW 0;	//COM.CODE
      CDB;	//ComDB->Instanz-DB
      UC    "GCS7_RS485Ctrl";	//Convert (CODE=DBW0)
      CDB;	//ElementDB->Instanz-DB
// Recipe Nr    
      L     4;	//*3.2* Character offset
      T     DBW 40;	//COM.Element.AddrOffset
      L     #InRecipeNr;
      T     DBD 36;	//COM.Element.InOutValue
      L     12;	//Convert DInt to 2-ASCII
      T     DBW 0;	//COM.CODE
      CDB;	//ComDB->Instanz-DB
      UC    "GCS7_RS485Ctrl";	//Convert (CODE=DBW0)
      CDB;	//ElementDB->Instanz-DB
//*3.2* Nominal Motor Current
      L     6;	//*3.2* Character offset
      T     DBW 40;	//COM.Element.AddrOffset
      L     #InMotorCurrent;
      T     DBD 36;	//COM.Element.InOutValue
      L     16;	//Convert DInt to 6-ASCII
      T     DBW 0;	//COM.CODE
      CDB;	//ComDB->Instanz-DB
      UC    "GCS7_RS485Ctrl";	//Convert (CODE=DBW0)
      CDB;	//ElementDB->Instanz-DB
//  
      L     20;	//Lenght in byte //[3.0]
      T     DBW 78;	//COM.Telegram.Len
      L     36;	//Lenght in byte
      T     DBW 86;	//COM.Telegram.LenAnswer
      JU    SndZ;
//======================================================================
//Answer Telegramm: Copy reveived data to element
//======================================================================
//--------------------
//Receive A 
//--------------------
Rcv:  R     #OutComFault;
      L     #tmpCommand;
      L     'A';
      <>I;
      JC    SAVE;
      AN    #Par.OutHelpFlags.OutFaultResetDone;
      JC    r_H1;
      S     #Par.OutHelpFlags.OutTestNewAlarm;
//StepNr
r_H1: L     2;	//Character offset
      T     DBW 40;	//COM.Element.AddrOffset
      L     22;	//Convert 2-ASCII to DInt
      T     DBW 0;	//COM.CODE
      CDB;	//ComDB->Instanz-DB
      UC    "GCS7_RS485Ctrl";	//Convert (CODE=DBW0)
      CDB;	//ElementDB->Instanz-DB
      L     DBD 36;	//COM.Element.InOutValue
      T     #OutLCStep;
//LC status
      L     0;	//Character offset
      T     DBW 40;	//COM.Element.AddrOffset
      L     42;	//Convert 2-ASCII to Hex
      T     DBW 0;	//COM.CODE
      CDB;	//ComDB->Instanz-DB
      UC    "GCS7_RS485Ctrl";	//Convert (CODE=DBW0)
      CDB;	//ElementDB->Instanz-DB
      L     DBD 36;	//COM.Element.InOutValue
      LAR1  P##tmpStatus_h;
      T     LB [AR1,P#0.0];	//-->tmpStatus_h
      A     #tmpStatus_h.Remote;
      =     #Par.Status.RemoteControl;
      A     #tmpStatus_h.InPosition;
      =     #Par.Status.InPosition;
      A     #tmpStatus_h.Operation;
      =     #Par.Status.Operation;
      A     #tmpStatus_h.Startupdone;	//*3.1* Added to check status bits
      =     #Par.Status.Startup;	//*3.1* Added to check status bits
      A     #tmpStatus_h.Level;	//*3.1* Added to check status bits
      =     #Par.Status.LevelProduct;	//*3.1* Added to check status bits
      A     #tmpStatus_h.WarningHLC;	//*3.1* Added to check status bits
      =     #Par.Status.WarningHLC;	//*3.1* Added to check status bits
      A     #tmpStatus_h.SumFault;
      =     #Par.Status.SumFault;
//Alarm number / LC alarm bit mask
      L     4;	//Character offset
      T     DBW 40;	//COM.Element.AddrOffset
      L     22;	//Convert 2-ASCII to DInt
      T     DBW 0;	//COM.CODE
      CDB;	//ComDB->Instanz-DB
      UC    "GCS7_RS485Ctrl";	//Convert (CODE=DBW0)
      CDB;	//ElementDB->Instanz-DB
      L     DBD 36;	//COM.Element.InOutValue
      T     #OutAlarmNr;
//*3.2* Actual Motor current
      L     6;	//Character offset
      T     DBW 40;	//COM.Element.AddrOffset
      L     26;	//Convert 6-ASCII to DInt
      T     DBW 0;	//COM.CODE
      CDB;	//ComDB->Instanz-DB
      UC    "GCS7_RS485Ctrl";	//Convert (CODE=DBW0)
      CDB;	//ElementDB->Instanz-DB
      L     DBD 36;	//COM.Element.InOutValue
      T     #OutCurrentMotorAc;	//*3.2*
//*3.2* Target Motor current
      L     12;	//*3.1* Character offset
      T     DBW 40;	//COM.Element.AddrOffset
      L     24;	//*3.1* Convert 4-ASCII to DInt
      T     DBW 0;	//COM.CODE
      CDB;	//ComDB->Instanz-DB
      UC    "GCS7_RS485Ctrl";	//Convert (CODE=DBW0)
      CDB;	//ElementDB->Instanz-DB
      L     DBD 36;	//COM.Element.InOutValue
      T     #OutCurrentMotorNom;	//*3.2*
//Weight
      L     16;	//*3.1* Character offset
      T     DBW 40;	//COM.Element.AddrOffset
      L     26;	//Convert 6-ASCII to DInt
      T     DBW 0;	//ERH.CODE
      CDB;	//ComDB->Instanz-DB
      UC    "GCS7_RS485Ctrl";	//Convert (CODE=DBW0)
      CDB;	//ElementDB->Instanz-DB
      L     DBD 36;	//ERH.Element.InOutValue
      T     #OutScaleWeight;
//*3.2* Actual Pressure
      L     22;	//*3.1* Character offset
      T     DBW 40;	//ERH.Element.AddrOffset
      L     24;	//Convert 4-ASCII to DInt
      T     DBW 0;	//ERH.CODE
      CDB;	//ComDB->Instanz-DB
      UC    "GCS7_RS485Ctrl";	//Convert (CODE=DBW0)
      CDB;	//ElementDB->Instanz-DB
      L     DBD 36;	//ERH.Element.InOutValue
      T     #OutPressure;	//*3.2*
//PMin
      L     26;	//*3.1* Character offset
      T     DBW 40;	//COM.Element.AddrOffset
      L     24;	//Convert 4-ASCII to DInt
      T     DBW 0;	//COM.CODE
      CDB;	//ComDB->Instanz-DB
      UC    "GCS7_RS485Ctrl";	//Convert (CODE=DBW0)
      CDB;	//ElementDB->Instanz-DB
      L     DBD 36;	//COM.Element.InOutValue
      T     #OutPMin;
//PMax
      L     30;	//*3.1* Character offset
      T     DBW 40;	//COM.Element.AddrOffset
      L     24;	//Convert 4-ASCII to DInt
      T     DBW 0;	//COM.CODE
      CDB;	//ComDB->Instanz-DB
      UC    "GCS7_RS485Ctrl";	//Convert (CODE=DBW0)
      CDB;	//ElementDB->Instanz-DB
      L     DBD 36;	//COM.Element.InOutValue
      T     #OutPMax;
//Recipe Nr 
      L     34;	//*3.1* Character offset
      T     DBW 40;	//COM.Element.AddrOffset
      L     22;	//Convert 2-ASCII to DInt
      T     DBW 0;	//COM.CODE
      CDB;	//ComDB->Instanz-DB
      UC    "GCS7_RS485Ctrl";	//Convert (CODE=DBW0)
      CDB;	//ElementDB->Instanz-DB
      L     DBD 36;	//COM.Element.InOutValue
      T     #OutRecipeNr;
      AN    #Par.Command.ResetAlarm;
      JC    tS1;
      S     #Par.OutHelpFlags.OutFaultResetDone;
tS1:  SET;
      R     #Par.OutHelpFlags.CmdFaultReset;
      R     #Par.Command.ResetAlarm;
      R     #Par.OutHelpFlags.CmdNewValue;
      JU    STOR;
SndZ: JU    STOR;
O22Z: NOP   0;
NETWORK
TITLE = PC Control
//=== Test Object number =====================
PC:   L     "SYS_DirectCtrlDB".PC.ObjectNo;	//PCControl.ObjectNo
      L     #Par.ParObjectNo;	//Input ObjectNo
      <>I;
      JC    Ctrl;
//=== Test OType      ========================
      L     1042;	//Input object type
      L     "SYS_DirectCtrlDB".PC.ObjectType;	//PCControl.ObjectType
      <>I;
      JC    Ctrl;
//=== Test Handshake =========================
      A     "SYS_DirectCtrlDB".PC.Hsk.FExamine;	//Handshake.FExamine
      JC    pExa;
      A     "SYS_DirectCtrlDB".PC.Hsk.FDefineCmd;	//Handshake.FDefineCmd
      JC    pCmd;
      A     "SYS_DirectCtrlDB".PC.Hsk.FDefinePara;	//Handshake.FDefinePara
      JC    pPar;
pIni: L     2;	//FcInit
      UC    "SYS_DirectCtrl";
      JU    Ctrl;
//Write parameter 
pPar: NOP   0;
//Write new commands from PC to Interface of group 
pCmd: A     "SYS_DirectCtrlDB".PC.Cmd1[4];	//Cmd1[4]  =CmdNewValue
      S     #CmdNewValue;
      A     "SYS_DirectCtrlDB".PC.Cmd1[8];	//Cmd1[8]  =CmdOff
      S     #CmdOff;
      A     "SYS_DirectCtrlDB".PC.Cmd1[9];	//Cmd1[9]  =CmdOn
      S     #CmdOn;
      A     "SYS_DirectCtrlDB".PC.Cmd1[10];	//Cmd1[10] =CmdNext
      S     #CmdNext;
      A     "SYS_DirectCtrlDB".PC.Cmd1[11];	//Cmd1[11] =CmdFaultReset
      S     #CmdFaultReset;
      A     "SYS_DirectCtrlDB".PC.Cmd1[13];	//Cmd1[13] =CmdManualOn
      S     #InManual;
      A     "SYS_DirectCtrlDB".PC.Cmd2[13];	//Cmd2[13] =CmdManualOff
      R     #InManual;
      A     "SYS_DirectCtrlDB".PC.Cmd1[14];	//Cmd1[14] =CmdReportOn
      S     #InReport;
      A     "SYS_DirectCtrlDB".PC.Cmd2[14];	//Cmd2[14] =CmdReportOff
      R     #InReport;
//Define Value
      AN    "SYS_DirectCtrlDB".PC.Hsk.FDefineValue;	// PC.Hsk.FDefineValue
      ON    #InManual;
      JC    pIni;
      LAR1  P#DBX 58.0;
      L     DBD [AR1,P#8.0];
      T     #InMotorCurrent;
      L     DBW [AR1,P#12.0];
      T     #InRecipeNr;
      L     DBD [AR1,P#14.0];
      T     #spare14;
      L     DBD [AR1,P#16.0];
      T     #OutCurrentMotorNom;
      JU    pIni;
pExa: TAR2;	//Address dynamic datas
      T     "SYS_DirectCtrlDB".GC.InDynAddr;	//-->PCControl.GC.InDynAddr
      L     #tmpLenDyn;	//Length dynamic datas
      T     "SYS_DirectCtrlDB".GC.InDynLen;	//-->PCControl.GC.InDynLen
      L     0;
      T     "SYS_DirectCtrlDB".GC.InParaAddr;	//-->PCControl.GC.InParaAddr
      T     "SYS_DirectCtrlDB".GC.InParaLen;	//-->PCControl.GC.InParaLen
      L     1;	//Code FcExamine
      UC    "SYS_DirectCtrl";
      L     10;	//Revision
      T     "SYS_DirectCtrlDB".GC.Revision;
Ctrl: NOP   0;
NETWORK
TITLE = [4.0] LCParameter
      L     #Par.ParObjectNo;
      L     "SYS_DirectCtrlLCDB".PC.ObjectNo;
      <>I;
      ON    #Par.ParOpto22;
      JC    LCP0;
      T     "SYS_DirectCtrlLCDB".GC.InObjectNo;
      L     #Par.ParComDB;
      T     "SYS_DirectCtrlLCDB".GC.InDBNr;
      L     #Par.ParLCAddr;
      T     "SYS_DirectCtrlLCDB".GC.InLCAddr;
LCP0: NOP   0;
NETWORK
TITLE =  Read LC data
      AN    #Par.ParOpto22;
      JC    O22A;
      OPN   DB [#tmpComDB];
      L     #Par.ParLCIdx;
      T     DBW 34;	//COM.Element.Index;
      L     1;	//Read LC data
      T     DBW 0;	//COM.CODE;
      CDB;
      UC    "GCS7_RS485Ctrl";
      CDB;
      L     #tmpFBNO;
      T     DBW 52;	//COM.LC0.FBNO;
      L     DINO;
      T     DBW 54;	//COM.LC0.DINO;
      TAR2  DBD 56;	//COM.LC0.AddrDyn;        
      L     0;
      T     DBD 60;	//COM.LC0.AddrPara;       
      L     #Par.ParLCAddr;
      T     DBD 64;	//COM.Telegram.LCAddr;
O22A: NOP   0;
NETWORK
TITLE = (Profibus) Read data and store Data 
      A     #Par.ParOpto22;
      JC    DP_A;
      L     #Par.ParIOByteNr;
      T     #tmpAddr;
      A     #InSimulation;
      JC    rSim;
      CALL  "SIEMENS_DPRD_DAT" (
           LADDR                    := #tmpAddr,
           RET_VAL                  := #tmpReturn,
           RECORD                   := #DPData);
      L     #tmpReturn;
      L     0;
      <>I;
      =     #Par.OutHelpFlags.OutComFaultRead;
      JC    rcv0;
      JU    rDP;
//read from Simulation
rSim: R     #Par.OutHelpFlags.OutComFaultRead;
      A     "GCS7_Gr_SimDPtoImage";
      L     P#I 0.0;
      JC    rDB1;
      OPN   "TEST_IOSimuliInput";
      L     P#DBX 0.0;
rDB1: L     #Par.ParIOByteNr;
      SLD   3;
      +D;
      LAR1;
      L     D [AR1,P#0.0];
      T     #DPData.StatusCommand;
      L     B [AR1,P#4.0];
      T     #DPData.NrSndDataSet;
      L     B [AR1,P#5.0];
      T     #DPData.IdxSndDataSet;
      L     B [AR1,P#6.0];
      T     #DPData.NrRcvDataSet;
      L     B [AR1,P#7.0];
      T     #DPData.IdxRcvDataSet;
      L     D [AR1,P#8.0];
      T     #DPData.Data[1];
      L     D [AR1,P#12.0];
      T     #DPData.Data[2];
      L     D [AR1,P#16.0];
      T     #DPData.Data[3];
      L     D [AR1,P#20.0];
      T     #DPData.Data[4];
//==Copy Status===============
rDP:  L     #DPData.NrRcvDataSet;
      L     0;
      ==I;
      JC    R001;
      CALL  "SIEMENS_BLKMOV" (
           SRCBLK                   := #DPData.StatusCommand,
           RET_VAL                  := #tmpReturn,
           DSTBLK                   := #Par.Status);
      AN    #Par.Status.NewRcvData;
      A     #InSimulation;
      JC    rcv0;
//===============================
//Answer Dataset 001
      L     #DPData.NrRcvDataSet;
      L     1;
      <>I;
      JC    r11;	//[4.0]
      CALL  "SIEMENS_BLKMOV" (
           SRCBLK                   := #DPData.Data,
           RET_VAL                  := #tmpReturn,
           DSTBLK                   := #Set001);
      L     #Set001.CurrentMotorNom;
      T     #OutCurrentMotorNom;
      L     #Set001.CurrentMotorAc;
      T     #OutCurrentMotorAc;
      L     #Set001.Pressure;
      T     #OutPressure;
      L     #Set001.PMin;
      T     #OutPMin;
      L     #Set001.PMax;
      T     #OutPMax;
      L     #Set001.RecipeNr;
      T     #OutRecipeNr;
      L     #Set001.Step;
      T     #OutLCStep;
//Reset old alarm flags with CmdFaultReset
      A     #Par.OutHelpFlags.OutFlagFaultResetDone;
      A     "SYS_Pulse1000ms";
      R     #Par.OutHelpFlags.OutFlagFaultResetDone;
      R     #Par.OutHelpFlags.OutFaultResetDone;
      S     #Par.OutHelpFlags.OutTestNewAlarm;
      L     0;
      L     #Set001.AlarmNr;
      ==I;
      =     #Par.OutHelpFlags.OutNoAlarm;
//  keep old alalrm number
      A     #Par.OutHelpFlags.OutNoAlarm;
      A     #Par.OutHelpFlags.OutRelevantFault;
      AN    #Par.OutHelpFlags.OutTestNewAlarm;
      AN    #InLocal;
      AN    #InManual;
      JC    rA1;
      T     #OutAlarmNr;
//--------------------------------------
//Calculate job weight on WtNotErasable
rA1:  JU    R11;	//[4.0]   
//===============================
//[4.0]--> LC Parameter 
//Reading dataset 11
R11:  L     "SYS_DirectCtrlLCDB".PC.ObjectNo;
      L     #Par.ParObjectNo;
      <>I;
      JC    R127;
      AN    "SYS_DirectCtrlLCDB".PC.Hsk.FExamineFirst;
      AN    "SYS_DirectCtrlLCDB".PC.Hsk.FExamineNext;
      JC    R127;
// -- Start Reading with Dataset 11
      L     11;
      T     #DPData.NrRcvDataSet;
      L     253;	//First
      A     "SYS_DirectCtrlLCDB".PC.Hsk.FExamineFirst;
      JC    rLC9;
      L     254;	//Next
rLC9: T     #DPData.IdxRcvDataSet;
      JU    rcv0;
//---Answer  dataset 11 ---
//---Answer  dataset 12 ---
r11:  L     #DPData.NrRcvDataSet;
      L     11;
      <>I;
      JC    rLCB;
// Answer Dataset 11
      L     '  ';
      T     "SYS_DirectCtrlLCDB".PC.Value[1];
      L     #DPData.Data[1];
      T     DB10.DBD 60;
      L     #DPData.Data[2];
      T     DB10.DBD 64;
      L     #DPData.Data[3];
      T     DB10.DBD 68;
      L     #DPData.Data[4];
      T     DB10.DBD 72;
      L     #DPData.IdxRcvDataSet;
      L     255;
      ==I;
      JC    rLCE;
      S     "SYS_DirectCtrlLCDB".GC.Set11Done;
      L     12;
      T     #DPData.NrRcvDataSet;
      L     0;
      T     #DPData.IdxRcvDataSet;
      JU    rcv0;	//--> Read dataset 12
// Answer Dataset 12
rLCB: L     #DPData.NrRcvDataSet;
      L     12;
      <>I;
      JC    r127;
      L     #DPData.Data[1];
      T     DB10.DBD 76;
      L     #DPData.Data[2];
      T     DB10.DBD 80;
      L     #DPData.Data[3];
      T     DB10.DBD 84;
      L     #DPData.Data[4];
      T     DB10.DBD 88;
      AN    "SYS_DirectCtrlLCDB".GC.Set11Done;
      JC    R127;
rLCE: L     12;
      CALL  "SYS_DirectCtrl";
      JU    R127;
//<--[4.0]
//===============================
//Answer  dataset 127
r127: L     #DPData.NrRcvDataSet;
      L     127;
      <>I;
      JC    r128;
      L     #DPData.Data[1];	//WtActual
      T     #OutScaleWeight;
      JU    R128;
//===============================
//Answer  dataset 128
r128: JU    r136;
//===============================
//Answer  dataset 136
r136: L     #DPData.NrRcvDataSet;
      L     136;
      <>I;
      JC    R001;	// =no valide answer read dataset 001
      JU    R001;
//===============================
//Read Dataset 001
R001: L     1;
      T     #DPData.NrRcvDataSet;
      L     0;
      T     #DPData.IdxRcvDataSet;
      A     #Par.OutHelpFlags.OutFaultResetDone;
      AN    "SYS_Pulse1000ms";
      S     #Par.OutHelpFlags.OutFlagFaultResetDone;
      JU    rcv0;
//===============================
//Read Dataset 127
R127: L     127;
      T     #DPData.NrRcvDataSet;
      L     0;
      T     #DPData.IdxRcvDataSet;
      JU    rcv0;
//===============================
//Read Dataset 128
R128: JU    R136;
//===============================
//Read Dataset 136
R136: JU    R001;
      JU    rcv0;
//===============================
rcv0: NOP   0;
DP_A: NOP   0;
NETWORK
TITLE = (Profibus) Status to ASW
      A     #Par.ParOpto22;
      JC    DP_E;
      A     #Par.OutHelpFlags.OutComFaultRead;
      O     #Par.OutHelpFlags.OutComFaultSend;
      =     #OutComFault;
//=======================================
//Init in local mode  
//=======================================
      AN    #InLocal;
      AN    #InManual;
      ON    #OutComFault;
      JC    alJL;
      L     0;
      T     #OutPressure;
alJL: NOP   0;
DP_E: NOP   0;
NETWORK
TITLE =  All State Init
//===Clear tmp Variable
//===Global Group Orders===
      A     "GCS7_Gr_OutManualOn";	//Global.OutManualOn
      S     #InManual;
      A     "GCS7_Gr_OutManualOff";	//Global.OutManualOff
      R     #InManual;
      A     #InManual;
      S     "GCS7_Gr_InManual";	//Global.InManualMode
//---Report is on---
      O     "GCS7_Gr_OutReportAll";	//---Global OutReportAll
      O     #InReport;
      =     #tmpReport;
//---FaultReset is on---
      A     "GCS7_Gr_OutFaultReset";	//GCS7_GR_OutFaultReset
      S     #CmdFaultReset;
//---Local---
      A     #InLocal;
      AN    #InManual;
      =     #tmpLocalFault;
      A     #tmpLocalFault;
      O     #InHWStop;
      O     #InDPFault;
      =     #tmpLocal;
//---Off---
      AN    #InManual;
      ON    #Par.ParManual;
      AN    #InEnable;
      O     #tmpLocal;
      O     #CmdOff;
      =     #tmpOff;
//---On---
      A     #CmdNext;
      AN    #InManual;
      O     #CmdOn;
      AN    #tmpOff;
      =     #tmpOn;
//--- Send Recipe
//--- Read Recipe
//--- tmpFault   
// Time out
      AN    #StStarting;
      AN    #StStopping;
      AN    #StFault;
      R     #Par.OutHelpFlags.OutAlarmTimeOut;
      JC    inJ1;
      A     #Par.OutHelpFlags.OutAlarmTimeOut;
      O     #StFault;
      JC    inJ1;
      L     0;
      L     #Par.OutMonTime;
      >I;
      =     #Par.OutHelpFlags.OutAlarmTimeOut;
      AN    "GCS7_Gr_OutTick200ms";	// Global Tick 200ms
      JC    inJ1;
      +     -2;	// Decrement all 200ms
      T     #Par.OutMonTime;
inJ1: NOP   0;
//=======================================
//Fault   
//=======================================
      LAR1  P##tmpFilter;
      L     #OutAlarmNr;
      +AR1;	//Pointer to #tmpFilter[OutAlarmNumber]
      L     #OutAlarmNr;
      L     0;
      <>I;
      AN    L [AR1,P#0.0];	//#tmpFilter[OutAlarmNumber]
      O;
      A     #Par.Status.SumFault;
      AN    #tmpFilter[0];
      =     #Par.OutHelpFlags.OutRelevantFault;
      A     #Par.Status.WrongValue;
      =     #OutWrongValue;
      A     #Par.OutHelpFlags.OutRelevantFault;
      O     #OutComFault;
      O     #Par.OutHelpFlags.OutAlarmTimeOut;
      O     #Par.Status.WrongValue;
      AN    #tmpLocal;
      =     #tmpFault;
NETWORK
TITLE = (Profibus) Prepare Command for MEAF
//================================
      A     #tmpOn;
      AN    #Par.OutHelpFlags.CmdNewValue;
      S     #Par.Command.Start;
      A     #StFault;
      A     #Par.OutHelpFlags.OutNoAlarm;
      O     #tmpOff;
      R     #Par.Command.Start;
//==============================
      A     #Par.ParOpto22;
      JC    DP_B;
//==============================
      A     #Par.Status.AcceptNewSendData;
      A     #Par.Command.ResetAlarm;
      R     #Par.Command.ResetAlarm;
      S     #Par.OutHelpFlags.OutFaultResetDone;
      A     #CmdFaultReset;
      AN    #Par.Status.AcceptNewSendData;
      R     #CmdFaultReset;
      S     #Par.Command.ResetAlarm;
      R     #Par.OutHelpFlags.OutAlarmTimeOut;
//==============================
      A     #Par.Status.NewDataReady;
      =     #Par.Command.AcceptNewDataReady;
//==============================
      SET;
      =     #Par.Command.CommandReady;
//==============================
      A     #Par.Status.NewRcvData;
      =     #Par.Command.AcceptNewRcvData;
//==============================
      AN    #Par.Status.AcceptNewSendData;
      =     #Par.Command.NewSendData;
DP_B: NOP   0;
NETWORK
TITLE = (Profibus) Send Data
      A     #Par.ParOpto22;
      JC    DP_C;
//======================================================
//Test Send Dataset 000 done
      L     #DPData.NrSndDataSet;
      L     0;
      <>I;
      JC    s128;
      JU    S128;	//-->send 128
//------------------------------------------------
//Test Send Dataset 128 done
s128: L     #DPData.NrSndDataSet;
      L     128;
      <>I;
      JC    s136;
      AN    #Par.Status.WrongValue;
      A     #Par.OutHelpFlags.CmdNewValue;
      A     #CmdNewValue;
      R     #Par.OutHelpFlags.CmdNewValue;
      R     #CmdNewValue;
      JU    S000;	//-->Send 136
//------------------------------------------------
//Test Send Dataset 136 done
s136: L     #DPData.NrSndDataSet;
      L     136;
      <>I;
      JC    S000;
      JU    S128;	//-->Send 128
//==================================================
//Send Dataset 128
S128: A     #CmdNewValue;
      =     #Par.OutHelpFlags.CmdNewValue;
      L     128;
      T     #DPData.NrSndDataSet;
      L     0;
      T     #DPData.IdxSndDataSet;
      L     #InMotorCurrent;
      SLD   16;
      T     #DPData.Data[1];
      L     0;
      T     #DPData.Data[2];
      T     #DPData.Data[3];
      L     #InRecipeNr;
      SLD   16;
      T     #DPData.Data[4];	//-->Byte 21
      JU    send;
//======================================================
//Send Dataset 0
S000: L     0;
      T     #DPData.NrSndDataSet;
      L     0;
      T     #DPData.IdxSndDataSet;
send: CALL  "SIEMENS_BLKMOV" (
           SRCBLK                   := #Par.Command,
           RET_VAL                  := #tmpReturn,
           DSTBLK                   := #DPData.StatusCommand);
      A     #InSimulation;
      JC    sSim;
      CALL  "SIEMENS_DPWR_DAT" (
           LADDR                    := #tmpAddr,
           RECORD                   := #DPData,
           RET_VAL                  := #tmpReturn);
      L     #tmpReturn;
      L     0;
      <>I;
      =     #Par.OutHelpFlags.OutComFaultSend;
      JU    DP_C;
//write to Simulation
sSim: R     #Par.OutHelpFlags.OutComFaultSend;
      A     "GCS7_Gr_SimDPtoImage";
      L     P#Q 0.0;
      JC    rDB2;
      OPN   "TEST_IOSimuliOutput";
      L     P#DBX 0.0;
rDB2: L     #Par.ParIOByteNr;
      SLD   3;
      +D;
      LAR1;
      L     #DPData.StatusCommand;
      T     D [AR1,P#0.0];
      L     #DPData.NrSndDataSet;
      T     B [AR1,P#4.0];
      L     #DPData.IdxSndDataSet;
      T     B [AR1,P#5.0];
      L     #DPData.NrRcvDataSet;
      T     B [AR1,P#6.0];
      L     #DPData.IdxRcvDataSet;
      T     B [AR1,P#7.0];
      L     #DPData.Data[1];
      T     D [AR1,P#8.0];
      L     #DPData.Data[2];
      T     D [AR1,P#12.0];
      L     #DPData.Data[3];
      T     D [AR1,P#16.0];
      L     #DPData.Data[4];
      T     D [AR1,P#20.0];
DP_C: NOP   0;
NETWORK
TITLE = States
//===State machine===
      A     #StStopped;
      JC    S0;
      A     #StStarting;
      JC    S1;
      A     #StStarted;
      JC    S2;
      A     #StStopping;
      JC    S3;
      A     #StFault;
      JC    S4;
      S     #StStopped;	//Init
      JU    S0;
NETWORK
TITLE =  StStopped
xxS0: S     #StStopped;
      R     #StStarted;
      JU    LOGX;
S0:   A     #tmpFault;
      R     #StStopped;
      JC    xxS4;	////--> Transition to StFault
      A     #tmpOn;
      R     #StStopped;
      JC    xxS1;	//--> Transition to StStarting
      JU    OUT;
NETWORK
TITLE =  StStarting
xxS1: S     #StStarting;
      R     #Par.OutHelpFlags.OutAlarmTimeOut;
      L     #Par.ParMonTime;
      T     #Par.OutMonTime;
      JU    OUT;
S1:   A     #tmpFault;	//Condition for StFault
      R     #StStarting;
      JC    xxS4;	//--> Transition to StFault
      A     #tmpOff;
      R     #StStarting;
      JC    xxS3;	//--> Transition to StStopping
      A     #Par.Status.Operation;
      R     #StStarting;
      JC    xxS2;	//--> Transition to StStarted
      JU    OUT;
NETWORK
TITLE =  StStarted
xxS2: S     #StStarted;
      JU    LOGX;
S2:   A     #tmpFault;	//Condition for StFault/StFalse
      R     #StStarted;
      JC    xxS4;	//--> Transition to StFault
      A     #tmpOff;
      ON    #Par.Status.Operation;
      R     #StStarted;
      JC    xxS3;	//--> Transition to StStopping
      JU    OUT;
NETWORK
TITLE =  StStopping
xxS3: S     #StStopping;
      R     #Par.OutHelpFlags.OutAlarmTimeOut;
      L     #Par.ParMonTime;
      T     #Par.OutMonTime;
      A     #StFault;
      R     #StFault;
      JC    LOGC;	//-->Message Operator ('fault cancelled' )
//State StStopping
S3:   A     #tmpFault;
      AN    #tmpLocal;
      R     #StStopping;
      JC    xxS4;	//-->Transition to StFault
      A     #tmpOn;
      R     #StStopping;
      JC    xxS1;	//-->Transition to StStarting 
      AN    #tmpFault;	//Transition to StFaulte
      AN    #Par.Status.Operation;
      R     #StStopping;
      JC    xxS0;	//-->Transition to StStopped 
      JU    OUT;
NETWORK
TITLE =  FAULT
// State Fault
S4:   AN    #tmpFault;	//---Condition for StStopping
      A     #Par.OutHelpFlags.OutTestNewAlarm;
      O     #tmpLocalFault;
      JC    xxS3;	// Transition to StStopping
      A     #Par.OutHelpFlags.OutTestNewAlarm;
      JC    xxS4;
      JU    OUT;
NETWORK
TITLE = LOG
xxS4: S     "GCS7_Gr_InFaultFlag";	//Gr.InFaultFlag
      S     #StFault;
      R     #Par.OutHelpFlags.OutFaultResetDone;
      R     #Par.OutHelpFlags.OutTestNewAlarm;
      CALL  "SYS_Horn_Code" (
           FcCode                   := 1,
           ParObjectType            := 1042,
           ParObjectNo              := #Par.ParObjectNo,
           ParHornCode              := #Par.ParHornCode);
      L     #Par.ParMonTime;
      T     #Par.OutMonTime;
//Alarm Communication
      L     B#(1, 96);
      A     #OutComFault;
      JC    LOG;
//Tiemout
      A     #Par.OutHelpFlags.OutAlarmTimeOut;
      L     B#(1, 94);	// Message ('fault timeout')
      JC    LOG;
//Alarm-Nr 1..80
      L     0;
      L     #OutAlarmNr;
      ==I;
      JC    LOG2;
      L     B#(1, 0);
      OW;
      JU    LOG;	//Alarms 1..80
//Fault Wrong Value
LOG2: A     #Par.Status.WrongValue;
      L     B#(1, 95);	// Message ('fault wrong value')
      JC    LOG;
//Collected Alarm
      L     B#(1, 99);	// Message ('fault collected alarm')
      JU    LOG;
//===============================================
//State Transition
LOGX: AN    #tmpReport;
      JC    OUT;
      A     #StStopped;
      L     B#(4, 91);	//Message ('Stopped')
      JC    LOG;
      A     #StStarted;
      L     B#(4, 92);	//Message ('Dosing')
      JC    LOG;
      JU    OUT;
LOGC: L     B#(4, 0);	//Message ('fault cancelled')
LOG:  A     #Par.ParLogOff;	//---Set LOG Message
      JC    SAVE;
      T     #tmpLOGvalue;
      L     W#16#FF;
      AW;
      T     #OutAlarmNrLog;
      CALL  "GCS7_LogConvert" (
           ObjectNo                 := #Par.ParObjectNo,
           MsgType                  := #Par.ParMsgType,
           ClassMsgTxt              := #tmpLOGvalue,
           OType                    := 1042);	//LOG Message Converter / Entry / Contains Class and TextNo
SAVE: NOP   0;
NETWORK
TITLE = (Opto22) Communication start
//Prepare Telegram for send
OUT:  AN    #Par.ParOpto22;
      JC    OUT2;
      A     DBX 50.0;	//COM.LC0.CmdPut
      O     DBX 50.1;	//COM.LC0.CmdGet
      JC    OUT2;
//--- 'A'
      A     #Par.Command.Start;
      =     #tmpFlag;
      A     #StStarting;
      O     #StStarted;
      AN    #tmpOff;
      AN    #tmpLocal;
      =     #Par.Command.Start;
      A     #CmdNewValue;
      AN    #Par.OutHelpFlags.CmdNewValue;
      R     #CmdNewValue;
      S     #Par.OutHelpFlags.CmdNewValue;
      A     #CmdFaultReset;
      R     #CmdFaultReset;
      S     #Par.Command.ResetAlarm;
      R     #Par.OutHelpFlags.OutAlarmTimeOut;
      L     'A';
      T     DBB 51;	//COM.LC0.Command;
      SET;
      S     DBX 50.0;	//COM.LC0.CmdPut 
NETWORK
TITLE = Global End
OUT2: A     #StStarted;
      O     #StStarting;
      AN    #tmpOff;
      AN    #tmpLocal;
      =     #OutpEnable;
      SET;	//---Clear all commands
      R     #CmdOff;
      R     #CmdOn;
      R     #CmdNext;
//--Output for group 
      AN    #InLocal;
      O     #InManual;
      A     #InDPFault;
      S     "GCS7_Gr_InDPFault";
      AN    #InLocal;
      O     #InManual;
      A     #InHWStop;
      S     "GCS7_Gr_InHWStop";
NETWORK
TITLE = State Code
//--Stopped, Substate ---
      AN    #StStopped;
      JC    STC2;
      L     41;	//Code: StStopped.HWStop
      A     #InHWStop;
      JC    STC;
      L     51;	//Code: StStopped.DPFault
      A     #InDPFault;
      JC    STC;
      L     1;	// Code: stopped
      JC    STC;
//--------------------
STC2: L     2;	//Code: StStarting
      A     #StStarting;
      JC    STC;
      L     3;	//Code: StStarted
      A     #StStarted;
      JC    STC;
      L     7;	//Code: StStopping
      A     #StStopping;
      JC    STC;
      L     32;	//Code: fault
STC:  L     #StCode;	//Old state code
      TAK;
      T     #StCode;	//Save state code
      <>I;
      L     3;	//Load code for CBit methode
      CC    "SYS_CBitCtrl";
NETWORK
TITLE =  Store LC data
      AN    #Par.ParOpto22;
      BEC;
      L     #Par.ParLCIdx;
      T     DBW 34;	//COM.Element.Index; 
      L     2;	//Store LC data
      T     DBW 0;	//COM.CODE;
      CDB;
      UC    "GCS7_RS485Ctrl";
      CDB;
STOR: BEU;
END_FUNCTION_BLOCK

